+-------------------+------------------+----------------------------+---------------------------+---------------------------------------+
| **value of data** | **size of data** | **value of dataToCompare** | **size of dataToCompare** | **CNM_ReturnTypes.ComparationResult** |
+===================+==================+============================+===========================+=======================================+
| null              | 0                | null                       | 0                         | EQUAL                                 |
+-------------------+------------------+----------------------------+---------------------------+---------------------------------------+
| null              | 0                | 16#01                      | 1                         | SMALLER                               |
+-------------------+------------------+----------------------------+---------------------------+---------------------------------------+
| 16#01             | 1                | null                       | 0                         | GREATER                               |
+-------------------+------------------+----------------------------+---------------------------+---------------------------------------+
| 16#00FF           | 2                | 16#FF                      | 1                         | EQUAL                                 |
+-------------------+------------------+----------------------------+---------------------------+---------------------------------------+
| 16#0100           | 2                | 16#FF                      | 1                         | GREATER                               |
+-------------------+------------------+----------------------------+---------------------------+---------------------------------------+
| 16#FF             | 1                | 16#0100                    | 2                         | SMALLER                               |
+-------------------+------------------+----------------------------+---------------------------+---------------------------------------+
| 16#FF             | 1                | 16#00FF                    | 2                         | EQUAL                                 |
+-------------------+------------------+----------------------------+---------------------------+---------------------------------------+
| 16#0FF0           | 2                | 16#F00F                    | 2                         | SMALLER                               |
+-------------------+------------------+----------------------------+---------------------------+---------------------------------------+

**Attention:** 
	Binary comparison means it compares values byte by byte, regardless of type information (signs, ``REAL`` etc...)
	and it compares padding bytes, too.

**Attention:** 
	``STRING`` and ``WSTRING`` is null terminated
	that means TwinCAT sets null byte/word at the end of the string and touches nothing else
	For example ``foo :STRING(3) := 'foo';`` looks binary 16#66 16#6F 16#6F 16#00.
	if you set foo to an empty string ``foo := ''`` it looks like 16#00 16#6F 16#6F 16#00.

**Attention:** 
	It works not for bits because the minimum size must be at least one byte. If the ``__SYSTEM.TYPE_CLASS``
	of ``data`` ``AND`` ``dataToCompare is ``__SYSTEM.TYPE_CLASS.TYPE_BOOL`` ``OR`` ``__SYSTEM.TYPE_CLASS.TYPE_BIT``
	it uses the ``TO_BOOL`` operator for comarison. That means for ``__SYSTEM.TYPE_CLASS.TYPE_BIT`` it has no idea
	if the single ``BIT`` is set or unset, it compares just the whole ``BYTE``.

.. <legal notes>

legal notes
=================
| SPDX-FileCopyrightText: © 2022 ekvip automation GmbH <info@ekvip.de>
| SPDX-License-Identifier: Apache-2.0
| For details check: Apache-2.0_

.. _Apache-2.0: https://www.apache.org/licenses/LICENSE-2.0

.. </legal notes>


:return: ``SMALLER``: ``data`` is smaller than ``dataToCompare``, 
``EQUAL``: ``data`` is equal to ``dataToCompare``,
``Greater``: ``data`` is greater to ``dataToCompare``

*)

{attribute 'analysis' := '-130'}
METHOD PROTECTED binaryCompare :CNM_ReturnTypes.ComparationResult
VAR_INPUT
	(* current binary data *)
	data			:ANY;
	(* binary data with smaller values *)
	dataToCompare	:ANY;
END_VAR
RETURN(THIS^.isDataNullOrSizeZero(data := data,dataToCompare := dataToCompare,result => binaryCompare));
IF (data.diSize < dataToCompare.diSize) THEN
	IF (THIS^.isDataZero(
		data := dataToCompare.pValue,
		size := dataToCompare.diSize,
		end := dataToCompare.diSize - data.diSize
	)) THEN
		binaryCompare := THIS^.compareData(
			data := data.pValue,
			dataToCompare := dataToCompare.pValue,
			size := data.diSize
		);
	ELSE
		binaryCompare := CNM_ReturnTypes.ComparationResult.SMALLER;
	END_IF
ELSIF (data.diSize > dataToCompare.diSize) THEN
	IF (THIS^.isDataZero(
		data := data.pValue,
		size := data.diSize,
		end := data.diSize - dataToCompare.diSize
	)) THEN
		binaryCompare := THIS^.compareData(
			data := data.pValue,
			dataToCompare := dataToCompare.pValue,
			size := dataToCompare.diSize
		);
	ELSE
		binaryCompare := CNM_ReturnTypes.ComparationResult.GREATER;
	END_IF
ELSIF (THIS^.isDataBoolOrBit(data := data, dataToCompare := dataToCompare)) THEN
	IF (TO_BOOL(data.pValue^) AND (NOT TO_BOOL(dataToCompare.pValue^))) THEN
		binaryCompare := CNM_ReturnTypes.ComparationResult.GREATER;
	ELSIF  ((NOT TO_BOOL(data.pValue^)) AND TO_BOOL(dataToCompare.pValue^)) THEN
		binaryCompare := CNM_ReturnTypes.ComparationResult.SMALLER;
	END_IF
ELSIF (data.diSize = dataToCompare.diSize) THEN
	binaryCompare := THIS^.compareData(
		data := data.pValue,
		dataToCompare := dataToCompare.pValue,
		size := data.diSize
	);
END_IF
END_METHOD

(*

## Short summary
This abstract property returns the class name of the concrete object, 
It's for debugging purpose

.. <legal notes>

legal notes
=================
| SPDX-FileCopyrightText: © 2022 ekvip automation GmbH <info@ekvip.de>
| SPDX-License-Identifier: Apache-2.0
| For details check: Apache-2.0_

.. _Apache-2.0: https://www.apache.org/licenses/LICENSE-2.0

.. </legal notes>

*)

PROPERTY className :CNM_AbstractObject.ClassName
GET
className := 'CNM_Assertor.BinaryAssertions';
END_GET
END_PROPERTY

(*

## Short summary
This method compares the data of two byte pointers. 
The table below shows with some examples how it works.

+-------------------+----------------------------+----------+---------------------------------------+
| **value of data** | **value of dataToCompare** | **size** | **CNM_ReturnTypes.ComparationResult** |
+===================+============================+==========+=======================================+
| 16#00FF           | 16#FF                      | 1        | EQUAL                                 |
+-------------------+----------------------------+----------+---------------------------------------+
| 16#0100           | 16#FF                      | 1        | SMALLER                               |
+-------------------+----------------------------+----------+---------------------------------------+
| 16#FF             | 16#0100                    | 1        | GREATER                               |
+-------------------+----------------------------+----------+---------------------------------------+
| 16#FF             | 16#00FF                    | 1        | EQUAL                                 |
+-------------------+----------------------------+----------+---------------------------------------+
| 16#0FF0           | 16#F00F                    | 1        | GREATER                               |
+-------------------+----------------------------+----------+---------------------------------------+
| 16#0FF0           | 16#F00F                    | 2        | SMALLER                               |
+-------------------+----------------------------+----------+---------------------------------------+

**Attention:** 
	Binary comparison means it compares values byte by byte, regardless of type information (signs, ``REAL`` etc...)
	and it compares padding bytes, too.

**Attention:** 
	``STRING`` and ``WSTRING`` is null terminated
	that means TwinCAT sets null byte/word at the end of the string and touches nothing else
	For example ``foo :STRING(3) := 'foo';`` looks binary 16#66 16#6F 16#6F 16#00.
	if you set foo to an empty string ``foo := ''`` it looks like 16#00 16#6F 16#6F 16#00.

.. <legal notes>

legal notes
=================
| SPDX-FileCopyrightText: © 2022 ekvip automation GmbH <info@ekvip.de>
| SPDX-License-Identifier: Apache-2.0
| For details check: Apache-2.0_

.. _Apache-2.0: https://www.apache.org/licenses/LICENSE-2.0

.. </legal notes>


:return: ``SMALLER``: ``data`` is smaller than ``dataToCompare``, 
``EQUAL``: ``data`` is equal to ``dataToCompare``,
``Greater``: ``data`` is greater to ``dataToCompare``

*)
{attribute 'analysis' := '-41, -130'}
METHOD PROTECTED compareBytewise :CNM_ReturnTypes.ComparationResult
VAR_INPUT
	(* current binary data *)
	data			:POINTER TO BYTE;
	(* current binary data to compare *)
	dataToCompare	:POINTER TO BYTE;
	(* size to compare in bytes, it must be smaller or equal to the smaller size of both data *)
	size			:DINT;
	(* last index to compare *)
	end				:LINT;
END_VAR
VAR
	(* index of the current address *)
	pointerIndex	:LINT;
END_VAR
compareBytewise := CNM_ReturnTypes.ComparationResult.EQUAL;
// memcmp is not used, as it compares from low to highbyte which contradicts the semantics of Numberdatatypes
FOR pointerIndex := (size-1) TO end BY THIS^.DIRECTION_LE DO
	IF (data[pointerIndex] < dataToCompare[pointerIndex]) THEN
		compareBytewise := CNM_ReturnTypes.ComparationResult.SMALLER;
		RETURN;
	ELSIF (data[pointerIndex] > dataToCompare[pointerIndex]) THEN
		compareBytewise := CNM_ReturnTypes.ComparationResult.GREATER;
		RETURN;
	END_IF
END_FOR;
END_METHOD

(*

## Short summary
This method comapres the data of two byte pointers.
It tries to compare registerwise if it makes sens (pointers are aligned and size big enough)
The table below shows with some examples how it works.

+-------------------+------------------+----------------------------+---------------------------+---------------------------------------+
| **value of data** | **size of data** | **value of dataToCompare** | **size of dataToCompare** | **CNM_ReturnTypes.ComparationResult** |
+===================+==================+============================+===========================+=======================================+
| 16#00FF           | 2                | 16#FF                      | 1                         | EQUAL                                 |
+-------------------+------------------+----------------------------+---------------------------+---------------------------------------+
| 16#0100           | 2                | 16#FF                      | 1                         | GREATER                               |
+-------------------+------------------+----------------------------+---------------------------+---------------------------------------+
| 16#FF             | 1                | 16#0100                    | 2                         | SMALLER                               |
+-------------------+------------------+----------------------------+---------------------------+---------------------------------------+
| 16#FF             | 1                | 16#00FF                    | 2                         | EQUAL                                 |
+-------------------+------------------+----------------------------+---------------------------+---------------------------------------+
| 16#0FF0           | 2                | 16#F00F                    | 2                         | SMALLER                               |
+-------------------+------------------+----------------------------+---------------------------+---------------------------------------+

**Attention:** 
	Binary comparison means it compares values byte by byte, regardless of type information (signs, ``REAL`` etc...)
	and it compares padding bytes, too.

**Attention:** 
	``STRING`` and ``WSTRING`` is null terminated
	that means TwinCAT sets null byte/word at the end of the string and touches nothing else
	For example ``foo :STRING(3) := 'foo';`` looks binary 16#66 16#6F 16#6F 16#00.
	if you set foo to an empty string ``foo := ''`` it looks like 16#00 16#6F 16#6F 16#00.

.. <legal notes>

legal notes
=================
| SPDX-FileCopyrightText: © 2022 ekvip automation GmbH <info@ekvip.de>
| SPDX-License-Identifier: Apache-2.0
| For details check: Apache-2.0_

.. _Apache-2.0: https://www.apache.org/licenses/LICENSE-2.0

.. </legal notes>


:return: ``SMALLER``: ``data`` is smaller than ``dataToCompare``, 
``EQUAL``: ``data`` is equal to ``dataToCompare``,
``Greater``: ``data`` is greater to ``dataToCompare``

*)

{attribute 'analysis' := '-130'}
METHOD PROTECTED compareData :CNM_ReturnTypes.ComparationResult
VAR_INPUT
	(* current binary data *)
	data			:POINTER TO BYTE;
	(* current binary data to compare *)
	dataToCompare	:POINTER TO BYTE;
	(* size to compare in bytes, it must be smaller or equal to the smaller size of both data *)
	size			:DINT;
END_VAR
VAR
	(* just a flag to store if both pointer addresses are aligned *)
	arePointersAligned			:BOOL;
	(* number of remaining bytes if it iterates regiterwise through the data*)
	remainingBytes				:DINT;
END_VAR
arePointersAligned := (THIS^.isPointerAligend(data) AND THIS^.isPointerAligend(dataToCompare));

IF (arePointersAligned AND (size >= THIS^.REGISTER_SIZE)) THEN
	remainingBytes := THIS^.getRemainingBytes(size);
	IF (remainingBytes > THIS^.ZERO_SIZE) THEN
		compareData := THIS^.compareBytewise(
			data := data,
			dataToCompare := dataToCompare,
			size := size,
			end := (size - remainingBytes)
		);
		RETURN (compareData <> CNM_ReturnTypes.ComparationResult.EQUAL);
	END_IF
	compareData := THIS^.compareRegisterwise(
		data := data,
		dataToCompare := dataToCompare,
		size := (size - remainingBytes)
	);	
ELSE	
	compareData := THIS^.compareBytewise(
		data := data,
		dataToCompare := dataToCompare,
		size := size,
		end := THIS^.FIRST_DATA
	);
END_IF
END_METHOD

(*

## Short summary
This method comapres the data of two byte pointers, but it iterates registerwise through the data.
The table below shows with some examples how it works.

+------------------------+----------------------------+----------+---------------------------------------+
|    **value of data**   | **value of dataToCompare** | **size** | **CNM_ReturnTypes.ComparationResult** |
+========================+============================+==========+=======================================+
| 16#00FF_FFFF_0000_FFFF | 16#00FF_FFFF_0000_FFFF     | 8        | EQUAL                                 |
+------------------------+----------------------------+----------+---------------------------------------+
| 16#00FF_FFFF_0000_FFFF | 16#80FF_FFFF_0000_FFFF     | 8        | SMALLER                               |
+------------------------+----------------------------+----------+---------------------------------------+
| 16#80FF_FFFF_0000_FFFF | 16#00FF_FFFF_0000_FFFF     | 8        | GREATER                               |
+------------------------+----------------------------+----------+---------------------------------------+
| 16#FFFF_FFFF_0000_FFFF | 16#FFFF_FFFF_0000_FFFF     | 8        | EQUAL                                 |
+------------------------+----------------------------+----------+---------------------------------------+
| 16#80FF_FFFF_0000_FFFF | 16#70FF_FFFF_FFFF_FFFF     | 8        | GREATER                               |
+------------------------+----------------------------+----------+---------------------------------------+
| 16#70FF_FFFF_FFFF_FFFF | 16#80FF_FFFF_0000_FFFF     | 8        | SMALLER                               |
+------------------------+----------------------------+----------+---------------------------------------+

**Attention:** 
	Binary comparison means it compares values register by register, regardless of type information (signs, ``REAL`` etc...)
	and it compares padding bytes, too.

**Attention:** 
	``STRING`` and ``WSTRING`` is null terminated
	that means TwinCAT sets null byte/word at the end of the string and touches nothing else
	For example ``foo :STRING(3) := 'foo';`` looks binary 16#66 16#6F 16#6F 16#00.
	if you set foo to an empty string ``foo := ''`` it looks like 16#00 16#6F 16#6F 16#00.

.. <legal notes>

legal notes
=================
| SPDX-FileCopyrightText: © 2022 ekvip automation GmbH <info@ekvip.de>
| SPDX-License-Identifier: Apache-2.0
| For details check: Apache-2.0_

.. _Apache-2.0: https://www.apache.org/licenses/LICENSE-2.0

.. </legal notes>


:return: ``SMALLER``: ``data`` is smaller than ``dataToCompare``, 
``EQUAL``: ``data`` is equal to ``dataToCompare``,
``Greater``: ``data`` is greater to ``dataToCompare``

*)

{attribute 'analysis' := '-41, -130'}
METHOD PROTECTED compareRegisterwise :CNM_ReturnTypes.ComparationResult
VAR_INPUT
	(* current binary data *)
	data			:POINTER TO __XWORD;
	(* current binary data to compare *)
	dataToCompare	:POINTER TO __XWORD;
	(* size to compare in bytes, size must be a muliple of register size *)
	size			:DINT;
END_VAR
VAR
	(* index of the current address *)
	pointerIndex	:LINT;
END_VAR
compareRegisterwise := CNM_ReturnTypes.ComparationResult.EQUAL;

FOR pointerIndex := (((size)/THIS^.REGISTER_SIZE)-1) TO THIS^.FIRST_DATA BY THIS^.DIRECTION_LE DO
	IF (data[pointerIndex] < dataToCompare[pointerIndex]) THEN
		compareRegisterwise := CNM_ReturnTypes.ComparationResult.SMALLER;
		RETURN;
	ELSIF (data[pointerIndex] > dataToCompare[pointerIndex]) THEN
		compareRegisterwise := CNM_ReturnTypes.ComparationResult.GREATER;
		RETURN;
	END_IF
END_FOR;
END_METHOD

(*

## Short summary
This method calculates the number of bytes that are remaining
if size is divided by register size.

.. <legal notes>

legal notes
=================
| SPDX-FileCopyrightText: © 2022 ekvip automation GmbH <info@ekvip.de>
| SPDX-License-Identifier: Apache-2.0
| For details check: Apache-2.0_

.. _Apache-2.0: https://www.apache.org/licenses/LICENSE-2.0

.. </legal notes>


:return: number of bytes that are remaining if it iterates registerwise through the data

*)

METHOD PROTECTED getRemainingBytes :DINT
VAR_INPUT
	(* size in bytes *)
	size			:DINT;
END_VAR
getRemainingBytes := (size MOD THIS^.REGISTER_SIZE);
END_METHOD

(*

## Short summary
This method checks if the current Data and DataToCompare are both either bools or bits.

.. <legal notes>

legal notes
=================
| SPDX-FileCopyrightText: © 2022 ekvip automation GmbH <info@ekvip.de>
| SPDX-License-Identifier: Apache-2.0
| For details check: Apache-2.0_

.. _Apache-2.0: https://www.apache.org/licenses/LICENSE-2.0

.. </legal notes>


:return: ``TRUE`` data and dataToCompare are both bool / bits, otherwise false

*)

METHOD PROTECTED isDataBoolOrBit : BOOL
VAR_INPUT
	(* current binary data *)
	data			:ANY;
	(* binary data with smaller values *)
	dataToCompare	:ANY;
END_VAR
VAR CONSTANT
	(* for boolens to figure out if the size exactly one byte *) 
	SIZE_OF_ONE_BYTE	:DINT := 1;
END_VAR
isDataBoolOrBit := ((
	data.diSize = SIZE_OF_ONE_BYTE
	) AND (
		dataToCompare.diSize = SIZE_OF_ONE_BYTE
	) AND ( 
		(data.TypeClass = TYPE_CLASS.TYPE_BOOL)
		OR 	(data.TypeClass = TYPE_CLASS.TYPE_BIT)
	) AND (
			(dataToCompare.TypeClass = TYPE_CLASS.TYPE_BOOL)
			OR (dataToCompare.TypeClass = TYPE_CLASS.TYPE_BIT)
	)
);
END_METHOD

(*

## Short summary
This method checks if the two given pointers have a valid address and the size of data is defined.

+-------------------+------------------+----------------------------+---------------------------+---------------------------------------+--------------------------+
| **value of data** | **size of data** | **value of dataToCompare** | **size of dataToCompare** | **CNM_ReturnTypes.ComparationResult** | **ReturnValue**		   |
+===================+==================+============================+===========================+=======================================+==========================+
| null              | *                | null                       | *                         | EQUAL                                 | TRUE					   |
+-------------------+------------------+----------------------------+---------------------------+---------------------------------------+--------------------------+
| *              	| 0                | *	                        | 0                         | EQUAL                                 | TRUE					   |
+-------------------+------------------+----------------------------+---------------------------+---------------------------------------+--------------------------+
| null              | *                | *                          | *                         | SMALLER                               | TRUE					   |
+-------------------+------------------+----------------------------+---------------------------+---------------------------------------+--------------------------+
| *                 | 0                | *                          | *                         | SMALLER                               | TRUE					   |
+-------------------+------------------+----------------------------+---------------------------+---------------------------------------+--------------------------+
| *                 | *                | null                       | *                         | GREATER                               | TRUE					   |
+-------------------+------------------+----------------------------+---------------------------+---------------------------------------+--------------------------+
| *                 | *                | *                          | 0                         | GREATER                               | TRUE					   |
+-------------------+------------------+----------------------------+---------------------------+---------------------------------------+--------------------------+
Otherwise: EQUAL, FALSE
( referes to something not null / <> 0)


legal notes
=================
| SPDX-FileCopyrightText: © 2025 ekvip automation GmbH <info@ekvip.de>
| SPDX-License-Identifier: Apache-2.0
| For details check: Apache-2.0_

.. _Apache-2.0: https://www.apache.org/licenses/LICENSE-2.0

.. </legal notes>


:return: consider table

*)

METHOD PROTECTED isDataNullOrSizeZero : BOOL
VAR_INPUT
	(* current binary data *)
	data			:ANY;
	(* binary data with smaller values *)
	dataToCompare	:ANY;
END_VAR
VAR_OUTPUT
	(*see table*)
	result: CNM_ReturnTypes.ComparationResult;
END_VAR
result := CNM_ReturnTypes.ComparationResult.EQUAL;
isDataNullOrSizeZero := TRUE;
RETURN ((data.pValue = THIS^.NULL_POINTER) AND (dataToCompare.pValue = THIS^.NULL_POINTER));
RETURN ((data.diSize = THIS^.ZERO_SIZE) AND (dataToCompare.diSize = THIS^.ZERO_SIZE));
IF (
	((data.pValue = THIS^.NULL_POINTER) AND (dataToCompare.pValue <> THIS^.NULL_POINTER))
	OR ((data.diSize = THIS^.ZERO_SIZE) AND (dataToCompare.diSize <> THIS^.ZERO_SIZE))
)THEN
	result := CNM_ReturnTypes.ComparationResult.SMALLER;
ELSIF (
	((data.pValue <> THIS^.NULL_POINTER) AND (dataToCompare.pValue = THIS^.NULL_POINTER))
	OR ((data.diSize <> THIS^.ZERO_SIZE) AND (dataToCompare.diSize = THIS^.ZERO_SIZE))
)THEN
	result := CNM_ReturnTypes.ComparationResult.GREATER;
ELSE
	isDataNullOrSizeZero := FALSE;
END_IF;
END_METHOD

(*

## Short summary
This method checks if the data of a pointer is zero through all bytes (``size-1``)

+------------------------+----------+---------+------------------+
|    **value of data**   | **size** | **end** | **return value** |
+========================+==========+=========+==================+
| 16#00FF_FFFF_0000_0000 | 8        | 7       | TRUE             |
+------------------------+----------+---------+------------------+
| 16#00FF_FFFF_0000_0000 | 8        | 6       | FALSE            |
+------------------------+----------+---------+------------------+
| 16#80FF_FFFF_0000_0000 | 8        | 7       | FALSE            |
+------------------------+----------+---------+------------------+
| 16#0000_0000_0000_FFFF | 8        | 2       | TRUE             |
+------------------------+----------+---------+------------------+
| 16#0000_0000_0000_FFFF | 8        | 1       | FALSE            |
+------------------------+----------+---------+------------------+
| 16#70FF_FFFF_FFFF_FFFF | 8        | 8       | TRUE             |
+------------------------+----------+---------+------------------+

.. <legal notes>

legal notes
=================
| SPDX-FileCopyrightText: © 2022 ekvip automation GmbH <info@ekvip.de>
| SPDX-License-Identifier: Apache-2.0
| For details check: Apache-2.0_

.. _Apache-2.0: https://www.apache.org/licenses/LICENSE-2.0

.. </legal notes>


:return: ``TRUE`` all bytes are zero, ``FALSE`` at least one byte isn't zero

*)

{attribute 'analysis' := '-130'}
METHOD PROTECTED isDataZero :BOOL
VAR_INPUT
	(* current binary data *)
	data			:POINTER TO BYTE;
	(* size to compare in bytes *)
	size			:DINT;
	(* last index to compare *)
	end				:LINT;	
END_VAR
VAR
	isPointerAligned			:BOOL;
	remainingBytes				:DINT;
END_VAR
isPointerAligned := THIS^.isPointerAligend(data);

IF (isPointerAligned AND_THEN ((size-end) >= THIS^.REGISTER_SIZE)) THEN
	remainingBytes := THIS^.getRemainingBytes(size);
	IF (remainingBytes > THIS^.ZERO_SIZE) THEN
		isDataZero := THIS^.isDataZeroBytewise(
			data := data,
			size := size,
			end := (size - remainingBytes)
		);
		RETURN (NOT isDataZero);
	END_IF
	isDataZero := THIS^.isDataZeroRegisterwise(
		data := data,
		size := (size - remainingBytes),
		end := end
	);	
ELSE	
	isDataZero := THIS^.isDataZeroBytewise(
		data := data,
		size := size,
		end := end
	);
END_IF;
END_METHOD

(*

## Short summary
This method checks if the data of a byte pointer is zero through all bytes form (``size-1``) to ``end``.
The table below shows how it works.

+------------------------+----------+---------+------------------+
|    **value of data**   | **size** | **end** | **return value** |
+========================+==========+=========+==================+
| 16#00FF_FFFF_0000_0000 | 8        | 7       | TRUE             |
+------------------------+----------+---------+------------------+
| 16#00FF_FFFF_0000_0000 | 8        | 6       | FALSE            |
+------------------------+----------+---------+------------------+
| 16#80FF_FFFF_0000_0000 | 8        | 7       | FALSE            |
+------------------------+----------+---------+------------------+
| 16#0000_0000_0000_FFFF | 8        | 2       | TRUE             |
+------------------------+----------+---------+------------------+
| 16#0000_0000_0000_FFFF | 8        | 1       | FALSE            |
+------------------------+----------+---------+------------------+
| 16#70FF_FFFF_FFFF_FFFF | 8        | 8       | TRUE             |
+------------------------+----------+---------+------------------+

.. <legal notes>

legal notes
=================
| SPDX-FileCopyrightText: © 2022 ekvip automation GmbH <info@ekvip.de>
| SPDX-License-Identifier: Apache-2.0
| For details check: Apache-2.0_

.. _Apache-2.0: https://www.apache.org/licenses/LICENSE-2.0

.. </legal notes>


:return: ``TRUE`` all bytes are zero, ``FALSE`` at least one byte isn't zero

*)

{attribute 'analysis' := '-130, -41'}
METHOD PROTECTED isDataZeroBytewise :BOOL
VAR_INPUT
	(* current binary data *)
	data			:POINTER TO BYTE;
	(* size to compare in bytes *)
	size			:DINT;
	(* last index to compare *)
	end				:LINT;
END_VAR
VAR
	(* index of the current address *)
	pointerIndex	:LINT;
END_VAR
VAR CONSTANT
	NULL			:BYTE := 16#00;
END_VAR
isDataZeroBytewise := TRUE;

FOR pointerIndex := (size-1) TO end BY THIS^.DIRECTION_LE DO
	IF (data[pointerIndex] <> NULL) THEN
		isDataZeroBytewise := FALSE;
		RETURN;
	END_IF
END_FOR;
END_METHOD

(*

## Short summary
This method checks if the data of a ``__XWORD pointer`` is zero
through all bytes form (``size-1``) to ``end``.

.. <legal notes>

legal notes
=================
| SPDX-FileCopyrightText: © 2022 ekvip automation GmbH <info@ekvip.de>
| SPDX-License-Identifier: Apache-2.0
| For details check: Apache-2.0_

.. _Apache-2.0: https://www.apache.org/licenses/LICENSE-2.0

.. </legal notes>


:return: ``TRUE`` all bytes are zero, ``FALSE`` at least one byte isn't zero

*)

{attribute 'analysis' := '-41, -130'}
METHOD PROTECTED isDataZeroRegisterwise :BOOL
VAR_INPUT
	(* current binary data *)
	data			:POINTER TO __XWORD;
	(* size to compare in bytes *)
	size			:DINT;
	(* last index to compare *)
	end				:LINT;
END_VAR
VAR
	(* index of the current address *)
	pointerIndex	:LINT;
END_VAR
VAR CONSTANT
	NULL			:__XWORD := 0;
END_VAR
isDataZeroRegisterwise := TRUE;

FOR pointerIndex := (size-1) TO end BY THIS^.DIRECTION_LE DO
	IF (data[pointerIndex] <> NULL) THEN
		isDataZeroRegisterwise := FALSE;
		RETURN;
	END_IF
END_FOR;
END_METHOD

(*

## Short summary
This assertion method checks if all bytes of memory of
``data`` and ``dataToCompare`` are equal

**Attention:** 
	Binary comparison means it compares values byte by byte, regardless of type information (signs, ``REAL`` etc...)
	and it compares padding bytes, too.

**Attention:** 
	``STRING`` and ``WSTRING`` is null terminated
	that means TwinCAT sets null byte/word at the end of the string and touches nothing else
	For example ``foo :STRING(3) := 'foo';`` looks binary 16#66 16#6F 16#6F 16#00.
	if you set foo to an empty string ``foo := ''`` it looks like 16#00 16#6F 16#6F 16#00.

**Attention:** 
	It works not for bits because the minimum size must be at least one byte. If the ``__SYSTEM.TYPE_CLASS``
	of ``data`` ``AND`` ``dataToCompare is ``__SYSTEM.TYPE_CLASS.TYPE_BOOL`` ``OR`` ``__SYSTEM.TYPE_CLASS.TYPE_BIT``
	it uses the ``TO_BOOL`` operator for comarison. That means for ``__SYSTEM.TYPE_CLASS.TYPE_BIT`` it has no idea
	if the single ``BIT`` is set or unset, it compares just the whole ``BYTE``.

.. <legal notes>

legal notes
=================
| SPDX-FileCopyrightText: © 2022 ekvip automation GmbH <info@ekvip.de>
| SPDX-License-Identifier: Apache-2.0
| For details check: Apache-2.0_

.. _Apache-2.0: https://www.apache.org/licenses/LICENSE-2.0

.. </legal notes>



*)

METHOD isEqualTo
VAR_INPUT
	(* current binary data *)
	data			:ANY;
	(* binary data with the expected values *)
	dataToCompare	:ANY;
	(* message if the assertion is false *)
	message			:AssertMessage;
END_VAR
IF (THIS^.binaryCompare(data, dataToCompare) <> CNM_ReturnTypes.ComparationResult.EQUAL) THEN
	THIS^.assertionWasWrong(message, THIS^.getDebugInfo('isEqualTo'));
END_IF
END_METHOD

(*

## Short summary
This assertion method checks the bytes of memory of
``data`` and ``dataToCompare`` if the content of the first unequal
``data`` byte is greater than the byte of ``dataToCompare``
the assertion is true. Direction of comaprison is little endian.

**Attention:** 
	Binary comparison means it compares values byte by byte, regardless of type information (signs, ``REAL`` etc...)
	and it compares padding bytes, too.

**Attention:** 
	``STRING`` and ``WSTRING`` is null terminated
	that means TwinCAT sets null byte/word at the end of the string and touches nothing else
	For example ``foo :STRING(3) := 'foo';`` looks binary 16#66 16#6F 16#6F 16#00.
	if you set foo to an empty string ``foo := ''`` it looks like 16#00 16#6F 16#6F 16#00.

**Attention:** 
	It works not for bits because the minimum size must be at least one byte. If the ``__SYSTEM.TYPE_CLASS``
	of ``data`` ``AND`` ``dataToCompare is ``__SYSTEM.TYPE_CLASS.TYPE_BOOL`` ``OR`` ``__SYSTEM.TYPE_CLASS.TYPE_BIT``
	it uses the ``TO_BOOL`` operator for comarison. That means for ``__SYSTEM.TYPE_CLASS.TYPE_BIT`` it has no idea
	if the single ``BIT`` is set or unset, it compares just the whole ``BYTE``.

.. <legal notes>

legal notes
=================
| SPDX-FileCopyrightText: © 2022 ekvip automation GmbH <info@ekvip.de>
| SPDX-License-Identifier: Apache-2.0
| For details check: Apache-2.0_

.. _Apache-2.0: https://www.apache.org/licenses/LICENSE-2.0

.. </legal notes>



*)

METHOD isGreaterThan
VAR_INPUT
	(* current binary data *)
	data			:ANY;
	(* binary data with smaller values *)
	dataToCompare	:ANY;
	(* message if the assertion is false *)
	message			:AssertMessage;
END_VAR
IF (THIS^.binaryCompare(data, dataToCompare) <> CNM_ReturnTypes.ComparationResult.GREATER) THEN
	THIS^.assertionWasWrong(message, THIS^.getDebugInfo('isGreaterThan'));
END_IF
END_METHOD

(*

## Short summary
This assertion method checks the bytes of memory of
``data`` and ``dataToCompare`` if the content of the first unequal
``data`` byte is less than the byte of ``dataToCompare``
the assertion is true. Direction of comaprison is little endian.

.. <legal notes>

**Attention:** 
	Binary comparison means it compares values byte by byte, regardless of type information (signs, ``REAL`` etc...)
	and it compares padding bytes, too.

**Attention:** 
	``STRING`` and ``WSTRING`` is null terminated
	that means TwinCAT sets null byte/word at the end of the string and touches nothing else
	For example ``foo :STRING(3) := 'foo';`` looks binary 16#66 16#6F 16#6F 16#00.
	if you set foo to an empty string ``foo := ''`` it looks like 16#00 16#6F 16#6F 16#00.

**Attention:** 
	It works not for bits because the minimum size must be at least one byte. If the ``__SYSTEM.TYPE_CLASS``
	of ``data`` ``AND`` ``dataToCompare is ``__SYSTEM.TYPE_CLASS.TYPE_BOOL`` ``OR`` ``__SYSTEM.TYPE_CLASS.TYPE_BIT``
	it uses the ``TO_BOOL`` operator for comarison. That means for ``__SYSTEM.TYPE_CLASS.TYPE_BIT`` it has no idea
	if the single ``BIT`` is set or unset, it compares just the whole ``BYTE``.

legal notes
=================
| SPDX-FileCopyrightText: © 2022 ekvip automation GmbH <info@ekvip.de>
| SPDX-License-Identifier: Apache-2.0
| For details check: Apache-2.0_

.. _Apache-2.0: https://www.apache.org/licenses/LICENSE-2.0

.. </legal notes>



*)

METHOD isLessThan
VAR_INPUT
	(* current binary data *)
	data			:ANY;
	(* binary data with greater values *)
	dataToCompare	:ANY;
	(* message if the assertion is false *)
	message			:AssertMessage;
END_VAR
IF (THIS^.binaryCompare(data, dataToCompare) <> CNM_ReturnTypes.ComparationResult.SMALLER) THEN
	THIS^.assertionWasWrong(message, THIS^.getDebugInfo('isLessThan'));
END_IF
END_METHOD

(*

## Short summary
This assertion method checks if minimal one byte of memory of
``data`` and ``dataToCompare`` is not equal

**Attention:** 
	Binary comparison means it compares values byte by byte, regardless of type information (signs, ``REAL`` etc...)
	and it compares padding bytes, too.

**Attention:** 
	``STRING`` and ``WSTRING`` is null terminated
	that means TwinCAT sets null byte/word at the end of the string and touches nothing else
	For example ``foo :STRING(3) := 'foo';`` looks binary 16#66 16#6F 16#6F 16#00.
	if you set foo to an empty string ``foo := ''`` it looks like 16#00 16#6F 16#6F 16#00.

**Attention:** 
	It works not for bits because the minimum size must be at least one byte. If the ``__SYSTEM.TYPE_CLASS``
	of ``data`` ``AND`` ``dataToCompare is ``__SYSTEM.TYPE_CLASS.TYPE_BOOL`` ``OR`` ``__SYSTEM.TYPE_CLASS.TYPE_BIT``
	it uses the ``TO_BOOL`` operator for comarison. That means for ``__SYSTEM.TYPE_CLASS.TYPE_BIT`` it has no idea
	if the single ``BIT`` is set or unset, it compares just the whole ``BYTE``.

.. <legal notes>

legal notes
=================
| SPDX-FileCopyrightText: © 2022 ekvip automation GmbH <info@ekvip.de>
| SPDX-License-Identifier: Apache-2.0
| For details check: Apache-2.0_

.. _Apache-2.0: https://www.apache.org/licenses/LICENSE-2.0

.. </legal notes>



*)

METHOD isNotEqualTo
VAR_INPUT
	(* current binary data *)
	data			:ANY;
	(* binary data with the unexpected values *)
	dataToCompare	:ANY;
	(* message if the assertion is false *)
	message			:AssertMessage;
END_VAR
IF (THIS^.binaryCompare(data, dataToCompare) = CNM_ReturnTypes.ComparationResult.EQUAL) THEN
	THIS^.assertionWasWrong(message, THIS^.getDebugInfo('isNotEqualTo'));
END_IF
END_METHOD

(*

## Short summary
This method checks if an address is aligned to a register

.. <legal notes>

legal notes
=================
| SPDX-FileCopyrightText: © 2022 ekvip automation GmbH <info@ekvip.de>
| SPDX-License-Identifier: Apache-2.0
| For details check: Apache-2.0_

.. _Apache-2.0: https://www.apache.org/licenses/LICENSE-2.0

.. </legal notes>


:return: ``TRUE`` pointer address **is** aligned to a register,
``FALSE`` pointer address **isn't** aligned to a register

*)

METHOD PROTECTED isPointerAligend :BOOL
VAR_INPUT
	(* address to check *)
	in :PVOID;
END_VAR
VAR CONSTANT
	(* 
	for 32 bit systems address is aligned if 2#111 is unset,
	for 64 bit systems address is aligned if 2#1111 is unset
	*)
	ALIGNMENT_MASK	:__XWORD := (SIZEOF(__XWORD)-1);
	(* just to check if relevant bits unset *)
	WELL_ALIGNED	:__XWORD := 0;
END_VAR
isPointerAligend := ((in AND ALIGNMENT_MASK) = WELL_ALIGNED);
END_METHOD

END_FUNCTION_BLOCK

// ---- Assertor/classes/AbstractAssertion.TcPOU
(*

## Short summary
This abstract class is for all the assertion classes to ease and unify
the callbacks

.. <legal notes>

legal notes
=================
| SPDX-FileCopyrightText: © 2022 ekvip automation GmbH <info@ekvip.de>
| SPDX-License-Identifier: Apache-2.0
| For details check: Apache-2.0_

.. _Apache-2.0: https://www.apache.org/licenses/LICENSE-2.0

.. </legal notes>



*)

{attribute 'reflection'}
FUNCTION_BLOCK INTERNAL ABSTRACT AbstractAssertion EXTENDS CNM_AbstractObject.Object IMPLEMENTS IAssertCallBackSetter
VAR
	(* the class that must be informed if an assertion is false *)
	callBack	:IAssertCallBack;
END_VAR

(*

## Short summary
This method is called if an assertion was ``FALSE``

.. <legal notes>

legal notes
=================
| SPDX-FileCopyrightText: © 2022 ekvip automation GmbH <info@ekvip.de>
| SPDX-License-Identifier: Apache-2.0
| For details check: Apache-2.0_

.. _Apache-2.0: https://www.apache.org/licenses/LICENSE-2.0

.. </legal notes>



*)

METHOD PROTECTED assertionWasWrong
VAR_INPUT
	(* alarm message *)
	message			:AssertMessage;
	(* debugging information *) 
	additionalText	:Tc2_System.T_MaxString;
END_VAR
IF (THIS^.isObjectValid(THIS^.callBack)) THEN
	THIS^.callBack.assertionWasWrong(
		caller			:= THIS^,
		message			:= message,
		additionalText	:= additionalText
	);
END_IF
END_METHOD

(*

## Short summary
This abstract property returns the class name of the concrete object, 
It's for debugging purpose

**Attention:** 
	For derivations: **It is necessary that this property is overridden by the concrete class**

.. <legal notes>

legal notes
=================
| SPDX-FileCopyrightText: © 2022 ekvip automation GmbH <info@ekvip.de>
| SPDX-License-Identifier: Apache-2.0
| For details check: Apache-2.0_

.. _Apache-2.0: https://www.apache.org/licenses/LICENSE-2.0

.. </legal notes>

*)

PROPERTY ABSTRACT className : CNM_AbstractObject.ClassName
GET
END_GET
END_PROPERTY

(*

## Short summary
This method returns a debug info string

.. <legal notes>

legal notes
=================
| SPDX-FileCopyrightText: © 2022 ekvip automation GmbH <info@ekvip.de>
| SPDX-License-Identifier: Apache-2.0
| For details check: Apache-2.0_

.. _Apache-2.0: https://www.apache.org/licenses/LICENSE-2.0

.. </legal notes>


:return: debug info string, it contains the caller method name and the class name. 
Format is ``'ClassName.methodName: Assertion was false'``

*)

METHOD PROTECTED getDebugInfo :Tc2_System.T_MaxString
VAR_INPUT
	(* name of the caller method *) 
	caller	:Tc2_System.T_MaxString;
END_VAR
getDebugInfo := Tc2_Standard.CONCAT(
	THIS^.className,
	Tc2_Standard.CONCAT(
		'.',
		Tc2_Standard.CONCAT(
			caller,
			': Assertion was false'
		)
	)
);
END_METHOD

(*

## Short summary
This methods is the setter for the callback class if an assertion was false

.. <legal notes>

legal notes
=================
| SPDX-FileCopyrightText: © 2022 ekvip automation GmbH <info@ekvip.de>
| SPDX-License-Identifier: Apache-2.0
| For details check: Apache-2.0_

.. _Apache-2.0: https://www.apache.org/licenses/LICENSE-2.0

.. </legal notes>



*)

METHOD setCallBack
VAR_INPUT
	(* the class that must be informed if an assertion is false *)
	callBack	:IAssertCallBack;  
END_VAR
THIS^.callBack := callBack;
END_METHOD

END_FUNCTION_BLOCK

// ---- Assertor/Assertions/BitNumberAssertions/Byte/classes/ByteAssertions.TcPOU
(*

## Short summary
This class provides assert statements for bytes.

.. <legal notes>

legal notes
=================
| SPDX-FileCopyrightText: © 2022 ekvip automation GmbH <info@ekvip.de>
| SPDX-License-Identifier: Apache-2.0
| For details check: Apache-2.0_

.. _Apache-2.0: https://www.apache.org/licenses/LICENSE-2.0

.. </legal notes>



*)

{attribute 'reflection'}
FUNCTION_BLOCK INTERNAL ByteAssertions EXTENDS AbstractAssertion IMPLEMENTS IByteAssertions
VAR
END_VAR
VAR CONSTANT
	(* least significant bit *)
	LSB	:BYTE := 16#01;
	(* most significant bit *)
	MSB :BYTE := 16#80;
END_VAR

(*

## Short summary
This assertion method checks if the result current value bitwise ``AND`` mask is equal to the expected value

.. <legal notes>

legal notes
=================
| SPDX-FileCopyrightText: © 2022 ekvip automation GmbH <info@ekvip.de>
| SPDX-License-Identifier: Apache-2.0
| For details check: Apache-2.0_

.. _Apache-2.0: https://www.apache.org/licenses/LICENSE-2.0

.. </legal notes>



*)

METHOD andMaskIsEqualTo
VAR_INPUT
	(* current value to check *)
	currentValue	:BYTE;
	(* 2nd operand for bitwise operation *)
	mask			:BYTE;
	(* expected result after masking *)
	expectedValue	:BYTE;
	(* message if the assertion is false *)
	message			:AssertMessage;
END_VAR
IF ((currentValue AND mask) <> expectedValue) THEN
	THIS^.assertionWasWrong(message, THIS^.getDebugInfo('andMaskIsEqualTo'));
END_IF
END_METHOD

(*

## Short summary
This assertion method checks if the result current value bitwise ``AND`` mask
is not equal to the unexpected value

.. <legal notes>

legal notes
=================
| SPDX-FileCopyrightText: © 2022 ekvip automation GmbH <info@ekvip.de>
| SPDX-License-Identifier: Apache-2.0
| For details check: Apache-2.0_

.. _Apache-2.0: https://www.apache.org/licenses/LICENSE-2.0

.. </legal notes>



*)

METHOD andMaskIsNotEqualTo
VAR_INPUT
	(* current value to check *)
	currentValue	:BYTE;
	(* 2nd operand for bitwise operation *)
	mask			:BYTE;
	(* unexpected result after masking *)
	unexpectedValue	:BYTE;
	(* message if the assertion is false *)
	message			:AssertMessage;
END_VAR
IF ((currentValue AND mask) = unexpectedValue) THEN
	THIS^.assertionWasWrong(message, THIS^.getDebugInfo('andMaskIsNotEqualTo'));
END_IF
END_METHOD

(*

## Short summary
This assertion method checks if the selected bit of current value
is equal to the expected value

.. <legal notes>

legal notes
=================
| SPDX-FileCopyrightText: © 2022 ekvip automation GmbH <info@ekvip.de>
| SPDX-License-Identifier: Apache-2.0
| For details check: Apache-2.0_

.. _Apache-2.0: https://www.apache.org/licenses/LICENSE-2.0

.. </legal notes>



*)

METHOD bitXIsEqualTo
VAR_INPUT
	(* current value to check *)
	currentValue	:BYTE;
	(* number of bit to check *)
	number			:BitNumberByte;
	(* expected value of bit *)
	expectedValue	:BOOL;
	(* message if the assertion is false *)
	message			:AssertMessage;
END_VAR
IF (
	TO_BOOL(
		TO_BYTE(SHL(THIS^.LSB, number))
		AND currentValue
	) <> expectedValue
) THEN
	THIS^.assertionWasWrong(message, THIS^.getDebugInfo('bitXIsEqualTo'));
END_IF
END_METHOD

(*

## Short summary
This assertion method checks if the selected bit of current value
is not equal to the unexpected value

.. <legal notes>

legal notes
=================
| SPDX-FileCopyrightText: © 2022 ekvip automation GmbH <info@ekvip.de>
| SPDX-License-Identifier: Apache-2.0
| For details check: Apache-2.0_

.. _Apache-2.0: https://www.apache.org/licenses/LICENSE-2.0

.. </legal notes>



*)

METHOD bitXIsNotEqualTo
VAR_INPUT
	(* current value to check *)
	currentValue	:BYTE;
	(* number of bit to check *)
	number			:BitNumberByte;
	(* unexpected value of bit *)
	unexpectedValue	:BOOL;
	(* message if the assertion is false *)
	message			:AssertMessage;
END_VAR
IF (
	TO_BOOL(
		TO_BYTE(SHL(THIS^.LSB, number))
		AND currentValue
	) = unexpectedValue
) THEN
	THIS^.assertionWasWrong(message, THIS^.getDebugInfo('bitXIsNotEqualTo'));
END_IF
END_METHOD

(*

## Short summary
This assertion method checks if the selected bit of current value
is set

.. <legal notes>

legal notes
=================
| SPDX-FileCopyrightText: © 2022 ekvip automation GmbH <info@ekvip.de>
| SPDX-License-Identifier: Apache-2.0
| For details check: Apache-2.0_

.. _Apache-2.0: https://www.apache.org/licenses/LICENSE-2.0

.. </legal notes>



*)

METHOD bitXIsSet
VAR_INPUT
	(* current value to check *)
	currentValue	:BYTE;
	(* number of bit to check *)
	number			:BitNumberByte;
	(* message if the assertion is false *)
	message			:AssertMessage;
END_VAR
IF (
	NOT TO_BOOL(
		TO_BYTE(SHL(THIS^.LSB, number))
		AND currentValue
	)
) THEN
	THIS^.assertionWasWrong(message, THIS^.getDebugInfo('bitXIsSet'));
END_IF
END_METHOD

(*

## Short summary
This assertion method checks if the selected bit of current value
is unset

.. <legal notes>

legal notes
=================
| SPDX-FileCopyrightText: © 2022 ekvip automation GmbH <info@ekvip.de>
| SPDX-License-Identifier: Apache-2.0
| For details check: Apache-2.0_

.. _Apache-2.0: https://www.apache.org/licenses/LICENSE-2.0

.. </legal notes>



*)

METHOD bitXIsUnset
VAR_INPUT
	(* current value to check *)
	currentValue	:BYTE;
	(* number of bit to check *)
	number			:BitNumberByte;
	(* message if the assertion is false *)
	message			:AssertMessage;
END_VAR
IF (
	TO_BOOL(
		TO_BYTE(SHL(THIS^.LSB, number))
		AND currentValue
	)
) THEN
	THIS^.assertionWasWrong(message, THIS^.getDebugInfo('bitXIsUnset'));
END_IF
END_METHOD

(*

## Short summary
This abstract property returns the class name of the concrete object, 
It's for debugging purpose

.. <legal notes>

legal notes
=================
| SPDX-FileCopyrightText: © 2022 ekvip automation GmbH <info@ekvip.de>
| SPDX-License-Identifier: Apache-2.0
| For details check: Apache-2.0_

.. _Apache-2.0: https://www.apache.org/licenses/LICENSE-2.0

.. </legal notes>

*)

PROPERTY className :CNM_AbstractObject.ClassName
GET
className := 'CNM_Assertor.ByteAssertions';
END_GET
END_PROPERTY

(*

## Short summary
This assertion method checks if the least significant bit of current value
is equal to the expected value

.. <legal notes>

legal notes
=================
| SPDX-FileCopyrightText: © 2022 ekvip automation GmbH <info@ekvip.de>
| SPDX-License-Identifier: Apache-2.0
| For details check: Apache-2.0_

.. _Apache-2.0: https://www.apache.org/licenses/LICENSE-2.0

.. </legal notes>



*)

METHOD lsbIsEqualTo
VAR_INPUT
	(* current value to check *)
	currentValue	:BYTE;
	(* expected value of lsb *)
	expectedValue	:BOOL;
	(* message if the assertion is false *)
	message			:AssertMessage;
END_VAR
IF (TO_BOOL(currentValue AND THIS^.LSB) <> expectedValue) THEN
	THIS^.assertionWasWrong(message, THIS^.getDebugInfo('lsbIsEqualTo'));
END_IF
END_METHOD

(*

## Short summary
This assertion method checks if the least significant bit of current value
is not equal to the unexpected value

.. <legal notes>

legal notes
=================
| SPDX-FileCopyrightText: © 2022 ekvip automation GmbH <info@ekvip.de>
| SPDX-License-Identifier: Apache-2.0
| For details check: Apache-2.0_

.. _Apache-2.0: https://www.apache.org/licenses/LICENSE-2.0

.. </legal notes>



*)

METHOD lsbIsNotEqualTo
VAR_INPUT
	(* current value to check *)
	currentValue	:BYTE;
	(* unexpected value of lsb *)
	unexpectedValue	:BOOL;
	(* message if the assertion is false *)
	message			:AssertMessage;
END_VAR
IF (TO_BOOL(currentValue AND THIS^.LSB) = unexpectedValue) THEN
	THIS^.assertionWasWrong(message, THIS^.getDebugInfo('lsbIsNotEqualTo'));
END_IF
END_METHOD

(*

## Short summary
This assertion method checks if the least significant bit of current value
is set

.. <legal notes>

legal notes
=================
| SPDX-FileCopyrightText: © 2022 ekvip automation GmbH <info@ekvip.de>
| SPDX-License-Identifier: Apache-2.0
| For details check: Apache-2.0_

.. _Apache-2.0: https://www.apache.org/licenses/LICENSE-2.0

.. </legal notes>



*)

METHOD lsbIsSet
VAR_INPUT
	(* current value to check *)
	currentValue	:BYTE;
	(* message if the assertion is false *)
	message			:AssertMessage;
END_VAR
IF (NOT TO_BOOL(currentValue AND THIS^.LSB)) THEN
	THIS^.assertionWasWrong(message, THIS^.getDebugInfo('lsbIsSet'));
END_IF
END_METHOD

(*

## Short summary
This assertion method checks if the least significant bit of current value
is unset

.. <legal notes>

legal notes
=================
| SPDX-FileCopyrightText: © 2022 ekvip automation GmbH <info@ekvip.de>
| SPDX-License-Identifier: Apache-2.0
| For details check: Apache-2.0_

.. _Apache-2.0: https://www.apache.org/licenses/LICENSE-2.0

.. </legal notes>



*)

METHOD lsbIsUnset
VAR_INPUT
	(* current value to check *)
	currentValue	:BYTE;
	(* message if the assertion is false *)
	message			:AssertMessage;
END_VAR
IF (TO_BOOL(currentValue AND THIS^.LSB)) THEN
	THIS^.assertionWasWrong(message, THIS^.getDebugInfo('lsbIsUnset'));
END_IF
END_METHOD

(*

## Short summary
This assertion method checks if the most significant bit of current value
is equal to the expected value

.. <legal notes>

legal notes
=================
| SPDX-FileCopyrightText: © 2022 ekvip automation GmbH <info@ekvip.de>
| SPDX-License-Identifier: Apache-2.0
| For details check: Apache-2.0_

.. _Apache-2.0: https://www.apache.org/licenses/LICENSE-2.0

.. </legal notes>



*)

METHOD msbIsEqualTo
VAR_INPUT
	(* current value to check *)
	currentValue	:BYTE;
	(* expected value of msb *)
	expectedValue	:BOOL;
	(* message if the assertion is false *)
	message			:AssertMessage;
END_VAR
IF (TO_BOOL(currentValue AND THIS^.MSB) <> expectedValue) THEN
	THIS^.assertionWasWrong(message, THIS^.getDebugInfo('msbIsEqualTo'));
END_IF
END_METHOD

(*

## Short summary
This assertion method checks if the most significant bit of current value
is not equal to the unexpected value

.. <legal notes>

legal notes
=================
| SPDX-FileCopyrightText: © 2022 ekvip automation GmbH <info@ekvip.de>
| SPDX-License-Identifier: Apache-2.0
| For details check: Apache-2.0_

.. _Apache-2.0: https://www.apache.org/licenses/LICENSE-2.0

.. </legal notes>



*)

METHOD msbIsNotEqualTo
VAR_INPUT
	(* current value to check *)
	currentValue	:BYTE;
	(* unexpected value of msb *)
	unexpectedValue	:BOOL;
	(* message if the assertion is false *)
	message			:AssertMessage;
END_VAR
IF (TO_BOOL(currentValue AND THIS^.MSB) = unexpectedValue) THEN
	THIS^.assertionWasWrong(message, THIS^.getDebugInfo('msbIsNotEqualTo'));
END_IF
END_METHOD

(*

## Short summary
This assertion method checks if the most significant bit of current value
is set

.. <legal notes>

legal notes
=================
| SPDX-FileCopyrightText: © 2022 ekvip automation GmbH <info@ekvip.de>
| SPDX-License-Identifier: Apache-2.0
| For details check: Apache-2.0_

.. _Apache-2.0: https://www.apache.org/licenses/LICENSE-2.0

.. </legal notes>



*)

METHOD msbIsSet
VAR_INPUT
	(* current value to check *)
	currentValue	:BYTE;
	(* message if the assertion is false *)
	message			:AssertMessage;
END_VAR
IF (NOT TO_BOOL(currentValue AND THIS^.MSB)) THEN
	THIS^.assertionWasWrong(message, THIS^.getDebugInfo('msbIsSet'));
END_IF
END_METHOD

(*

## Short summary
This assertion method checks if the most significant bit of current value
is unset

.. <legal notes>

legal notes
=================
| SPDX-FileCopyrightText: © 2022 ekvip automation GmbH <info@ekvip.de>
| SPDX-License-Identifier: Apache-2.0
| For details check: Apache-2.0_

.. _Apache-2.0: https://www.apache.org/licenses/LICENSE-2.0

.. </legal notes>



*)

METHOD msbIsUnset
VAR_INPUT
	(* current value to check *)
	currentValue	:BYTE;
	(* message if the assertion is false *)
	message			:AssertMessage;
END_VAR
IF (TO_BOOL(currentValue AND THIS^.MSB)) THEN
	THIS^.assertionWasWrong(message, THIS^.getDebugInfo('msbIsUnset'));
END_IF
END_METHOD

(*

## Short summary
This assertion method checks if the result current value bitwise ``OR`` mask is equal to the expected value

.. <legal notes>

legal notes
=================
| SPDX-FileCopyrightText: © 2022 ekvip automation GmbH <info@ekvip.de>
| SPDX-License-Identifier: Apache-2.0
| For details check: Apache-2.0_

.. _Apache-2.0: https://www.apache.org/licenses/LICENSE-2.0

.. </legal notes>



*)

METHOD orMaskIsEqualTo
VAR_INPUT
	(* current value to check *)
	currentValue	:BYTE;
	(* 2nd operand for bitwise operation *)
	mask			:BYTE;
	(* expected result after masking *)
	expectedValue	:BYTE;
	(* message if the assertion is false *)
	message			:AssertMessage;
END_VAR
IF ((currentValue OR mask) <> expectedValue) THEN
	THIS^.assertionWasWrong(message, THIS^.getDebugInfo('orMaskIsEqualTo'));
END_IF
END_METHOD

(*

## Short summary
This assertion method checks if the result current value bitwise ``OR`` mask 
is not equal to the unexpected value

.. <legal notes>

legal notes
=================
| SPDX-FileCopyrightText: © 2022 ekvip automation GmbH <info@ekvip.de>
| SPDX-License-Identifier: Apache-2.0
| For details check: Apache-2.0_

.. _Apache-2.0: https://www.apache.org/licenses/LICENSE-2.0

.. </legal notes>



*)

METHOD orMaskIsNotEqualTo
VAR_INPUT
	(* current value to check *)
	currentValue	:BYTE;
	(* 2nd operand for bitwise operation *)
	mask			:BYTE;
	(* unexpected result after masking *)
	unexpectedValue	:BYTE;
	(* message if the assertion is false *)
	message			:AssertMessage;
END_VAR
IF ((currentValue OR mask) = unexpectedValue) THEN
	THIS^.assertionWasWrong(message, THIS^.getDebugInfo('orMaskIsNotEqualTo'));
END_IF
END_METHOD

(*

## Short summary
This assertion method checks if the current value is equal to the expected value

.. <legal notes>

legal notes
=================
| SPDX-FileCopyrightText: © 2022 ekvip automation GmbH <info@ekvip.de>
| SPDX-License-Identifier: Apache-2.0
| For details check: Apache-2.0_

.. _Apache-2.0: https://www.apache.org/licenses/LICENSE-2.0

.. </legal notes>



*)

METHOD valueIsEqualTo
VAR_INPUT
	(* current value to check *)
	currentValue	:BYTE;
	(* expected value to compare *)
	expectedValue	:BYTE;
	(* message if the assertion is false *)
	message			:AssertMessage;
END_VAR
IF (currentValue <> expectedValue) THEN
	THIS^.assertionWasWrong(message, THIS^.getDebugInfo('valueIsEqualTo'));
END_IF
END_METHOD

(*

## Short summary
This assertion method checks if the current value is greater than the less value

.. <legal notes>

legal notes
=================
| SPDX-FileCopyrightText: © 2022 ekvip automation GmbH <info@ekvip.de>
| SPDX-License-Identifier: Apache-2.0
| For details check: Apache-2.0_

.. _Apache-2.0: https://www.apache.org/licenses/LICENSE-2.0

.. </legal notes>



*)

METHOD valueIsGreaterThan
VAR_INPUT
	(* current value to check *)
	currentValue	:BYTE;
	(* less than lower limit *)
	lessValue		:BYTE;
	(* message if the assertion is false *)
	message			:AssertMessage;
END_VAR
IF (currentValue <= lessValue) THEN
	THIS^.assertionWasWrong(message, THIS^.getDebugInfo('valueIsGreaterThan'));
END_IF
END_METHOD

(*

## Short summary
This assertion method checks if the current value is inside a limit

**Attention:** 
	limits are included: ``valueIsInRangeOf(3, 3, 3)`` is a true assertion

.. <legal notes>

legal notes
=================
| SPDX-FileCopyrightText: © 2022 ekvip automation GmbH <info@ekvip.de>
| SPDX-License-Identifier: Apache-2.0
| For details check: Apache-2.0_

.. _Apache-2.0: https://www.apache.org/licenses/LICENSE-2.0

.. </legal notes>



*)

METHOD valueIsInRangeOf
VAR_INPUT
	(* lower limit for the current value *)
	lowerLimit		:BYTE;
	(* current value to check *)
	currentValue	:BYTE;
	(* upper limit for the current value *)
	upperLimit		:BYTE;
	(* message if the assertion is false *)
	message			:AssertMessage;
END_VAR
IF (
	(currentValue < lowerLimit)
	OR (currentValue > upperLimit)
) THEN
	THIS^.assertionWasWrong(message, THIS^.getDebugInfo('valueIsInRangeOf'));
END_IF
END_METHOD

(*

## Short summary
This assertion method checks if the current value is less than the greater value

.. <legal notes>

legal notes
=================
| SPDX-FileCopyrightText: © 2022 ekvip automation GmbH <info@ekvip.de>
| SPDX-License-Identifier: Apache-2.0
| For details check: Apache-2.0_

.. _Apache-2.0: https://www.apache.org/licenses/LICENSE-2.0

.. </legal notes>



*)

METHOD valueIsLessThan
VAR_INPUT
	(* current value to check *)
	currentValue	:BYTE;
	(* greater than upper limit *)
	greaterValue	:BYTE;
	(* message if the assertion is false *)
	message			:AssertMessage;
END_VAR
IF (currentValue >= greaterValue) THEN
	THIS^.assertionWasWrong(message, THIS^.getDebugInfo('valueIsLessThan'));
END_IF
END_METHOD

(*

## Short summary
This assertion method checks if the current value is less than or equal to the maximum value

.. <legal notes>

legal notes
=================
| SPDX-FileCopyrightText: © 2022 ekvip automation GmbH <info@ekvip.de>
| SPDX-License-Identifier: Apache-2.0
| For details check: Apache-2.0_

.. _Apache-2.0: https://www.apache.org/licenses/LICENSE-2.0

.. </legal notes>



*)

METHOD valueIsMax
VAR_INPUT
	(* current value to check *)
	currentValue	:BYTE;
	(* upper limit for the current value *)
	maximumValue	:BYTE;
	(* message if the assertion is false *)
	message			:AssertMessage;
END_VAR
IF (currentValue > maximumValue) THEN
	THIS^.assertionWasWrong(message, THIS^.getDebugInfo('valueIsMax'));
END_IF
END_METHOD

(*

## Short summary
This assertion method checks if the current value is greater than or equal to the minimum value

.. <legal notes>

legal notes
=================
| SPDX-FileCopyrightText: © 2022 ekvip automation GmbH <info@ekvip.de>
| SPDX-License-Identifier: Apache-2.0
| For details check: Apache-2.0_

.. _Apache-2.0: https://www.apache.org/licenses/LICENSE-2.0

.. </legal notes>



*)

METHOD valueIsMin
VAR_INPUT
	(* current value to check *)
	currentValue	:BYTE;
	(* lower limit for the current value *)
	minimumValue	:BYTE;
	(* message if the assertion is false *)
	message			:AssertMessage;
END_VAR
IF (currentValue < minimumValue) THEN
	THIS^.assertionWasWrong(message, THIS^.getDebugInfo('valueIsMin'));
END_IF
END_METHOD

(*

## Short summary
This assertion method checks if the current value is not equal to the unexpected value

.. <legal notes>

legal notes
=================
| SPDX-FileCopyrightText: © 2022 ekvip automation GmbH <info@ekvip.de>
| SPDX-License-Identifier: Apache-2.0
| For details check: Apache-2.0_

.. _Apache-2.0: https://www.apache.org/licenses/LICENSE-2.0

.. </legal notes>



*)

METHOD valueIsNotEqualTo
VAR_INPUT
	(* current value to check *)
	currentValue	:BYTE;
	(* unexpected value to compare *)
	unexpectedValue	:BYTE;
	(* message if the assertion is false *)
	message			:AssertMessage;
END_VAR
IF (currentValue = unexpectedValue) THEN
	THIS^.assertionWasWrong(message, THIS^.getDebugInfo('valueIsNotEqualTo'));
END_IF
END_METHOD

(*

## Short summary
This assertion method checks if the result current value bitwise ``XOR`` mask is equal to the expected value

.. <legal notes>

legal notes
=================
| SPDX-FileCopyrightText: © 2022 ekvip automation GmbH <info@ekvip.de>
| SPDX-License-Identifier: Apache-2.0
| For details check: Apache-2.0_

.. _Apache-2.0: https://www.apache.org/licenses/LICENSE-2.0

.. </legal notes>



*)

METHOD xorMaskIsEqualTo
VAR_INPUT
	(* current value to check *)
	currentValue	:BYTE;
	(* 2nd operand for bitwise operation *)
	mask			:BYTE;
	(* expected result after masking *)
	expectedValue	:BYTE;
	(* message if the assertion is false *)
	message			:AssertMessage;
END_VAR
IF ((currentValue XOR mask) <> expectedValue) THEN
	THIS^.assertionWasWrong(message, THIS^.getDebugInfo('xorMaskIsEqualTo'));
END_IF
END_METHOD

(*

## Short summary
This assertion method checks if the result current value bitwise ``XOR`` mask 
is not equal to the unexpected value

.. <legal notes>

legal notes
=================
| SPDX-FileCopyrightText: © 2022 ekvip automation GmbH <info@ekvip.de>
| SPDX-License-Identifier: Apache-2.0
| For details check: Apache-2.0_

.. _Apache-2.0: https://www.apache.org/licenses/LICENSE-2.0

.. </legal notes>



*)

METHOD xorMaskIsNotEqualTo
VAR_INPUT
	(* current value to check *)
	currentValue	:BYTE;
	(* 2nd operand for bitwise operation *)
	mask			:BYTE;
	(* unexpected result after masking *)
	unexpectedValue	:BYTE;
	(* message if the assertion is false *)
	message			:AssertMessage;
END_VAR
IF ((currentValue XOR mask) = unexpectedValue) THEN
	THIS^.assertionWasWrong(message, THIS^.getDebugInfo('xorMaskIsNotEqualTo'));
END_IF
END_METHOD

END_FUNCTION_BLOCK

// ---- Assertor/Assertions/BitNumberAssertions/classes/BitNumberAssertions.TcPOU
(*

## Short summary

 This class provides assert statements for bit numbers:
 It implements the interface `IBitNumberAssertions`
 For ``BYTE`` use `BitNumberAssertions.short`
 For ``WORD`` use `BitNumberAssertions.simple`
 For ``DWORD`` use `BitNumberAssertions.double`
 For ``LWORD`` use `BitNumberAssertions.long`
 For ``__XWORD`` use `BitNumberAssertions.x`

.. <legal notes>

legal notes
=================
| SPDX-FileCopyrightText: © 2022 ekvip automation GmbH <info@ekvip.de>
| SPDX-License-Identifier: Apache-2.0
| For details check: Apache-2.0_

.. _Apache-2.0: https://www.apache.org/licenses/LICENSE-2.0

.. </legal notes>



*)

{attribute 'reflection'}
FUNCTION_BLOCK INTERNAL BitNumberAssertions 
EXTENDS CNM_AbstractObject.Object 
IMPLEMENTS IBitNumberAssertions, IAssertCallBacksetter
VAR
	(* class to handle byte assertions *)
	byteAssertions	:ByteAssertions();
	(* class to handle word assertions *)
	wordAssertions	:WordAssertions();
	(* class to handle dword assertions *)
	dwordAssertions	:DWordAssertions();
	(* class to handle lword assertions *)
	lwordAssertions	:LWordAssertions();
	(* class to handle xword assertions *)
	xwordAssertions	:XWordAssertions();
END_VAR

(*

## Short summary
This abstract property returns the class name of the concrete object, 
It's for debugging purpose

.. <legal notes>

legal notes
=================
| SPDX-FileCopyrightText: © 2022 ekvip automation GmbH <info@ekvip.de>
| SPDX-License-Identifier: Apache-2.0
| For details check: Apache-2.0_

.. _Apache-2.0: https://www.apache.org/licenses/LICENSE-2.0

.. </legal notes>

*)

PROPERTY className :CNM_AbstractObject.ClassName
GET
className := 'CNM_Assertor.BitNumberAssertions';
END_GET
END_PROPERTY

(*

## Short summary
Returns the interface `IDwordAssertions`
with assert statements for double words ``DWORD`` 

.. <legal notes>

legal notes
=================
| SPDX-FileCopyrightText: © 2022 ekvip automation GmbH <info@ekvip.de>
| SPDX-License-Identifier: Apache-2.0
| For details check: Apache-2.0_

.. _Apache-2.0: https://www.apache.org/licenses/LICENSE-2.0

.. </legal notes>

*)

PROPERTY double :IDwordAssertions
GET
double := THIS^.dwordAssertions;
END_GET
END_PROPERTY

(*

## Short summary
Returns the interface `ILwordAssertions`
with assert statements for long words ``LWORD`` 

.. <legal notes>

legal notes
=================
| SPDX-FileCopyrightText: © 2022 ekvip automation GmbH <info@ekvip.de>
| SPDX-License-Identifier: Apache-2.0
| For details check: Apache-2.0_

.. _Apache-2.0: https://www.apache.org/licenses/LICENSE-2.0

.. </legal notes>

*)

PROPERTY long :ILwordAssertions
GET
long := THIS^.lwordAssertions;
END_GET
END_PROPERTY

(*

## Short summary
This methods is the setter for the callback class if an assertion was false

.. <legal notes>

legal notes
=================
| SPDX-FileCopyrightText: © 2022 ekvip automation GmbH <info@ekvip.de>
| SPDX-License-Identifier: Apache-2.0
| For details check: Apache-2.0_

.. _Apache-2.0: https://www.apache.org/licenses/LICENSE-2.0

.. </legal notes>



*)

METHOD setCallBack
VAR_INPUT
	(* the class that must be informed if an assertion is false *)
	callBack	:IAssertCallBack;  
END_VAR
THIS^.byteAssertions.setCallBack(callBack);
THIS^.wordAssertions.setCallBack(callBack);
THIS^.dwordAssertions.setCallBack(callBack);
THIS^.lwordAssertions.setCallBack(callBack);
THIS^.xwordAssertions.setCallBack(callBack);
END_METHOD

(*

## Short summary
Returns the interface `IByteAssertions`
with assert statements for bytes

.. <legal notes>

legal notes
=================
| SPDX-FileCopyrightText: © 2022 ekvip automation GmbH <info@ekvip.de>
| SPDX-License-Identifier: Apache-2.0
| For details check: Apache-2.0_

.. _Apache-2.0: https://www.apache.org/licenses/LICENSE-2.0

.. </legal notes>

*)

PROPERTY short :IByteAssertions
GET
short := THIS^.byteAssertions;
END_GET
END_PROPERTY

(*

## Short summary
Returns the interface `IWordAssertions`
with assert statements for words 

.. <legal notes>

legal notes
=================
| SPDX-FileCopyrightText: © 2022 ekvip automation GmbH <info@ekvip.de>
| SPDX-License-Identifier: Apache-2.0
| For details check: Apache-2.0_

.. _Apache-2.0: https://www.apache.org/licenses/LICENSE-2.0

.. </legal notes>

*)

PROPERTY simple :IWordAssertions
GET
simple := THIS^.wordAssertions;
END_GET
END_PROPERTY

(*

## Short summary
Returns the interface `IXwordAssertions`
with assert statements for register length words ``__XWORD``

.. <legal notes>

legal notes
=================
| SPDX-FileCopyrightText: © 2022 ekvip automation GmbH <info@ekvip.de>
| SPDX-License-Identifier: Apache-2.0
| For details check: Apache-2.0_

.. _Apache-2.0: https://www.apache.org/licenses/LICENSE-2.0

.. </legal notes>

*)

PROPERTY x :IXwordAssertions
GET
x := THIS^.xwordAssertions;
END_GET
END_PROPERTY

END_FUNCTION_BLOCK

// ---- Assertor/Assertions/BitNumberAssertions/Word/classes/WordAssertions.TcPOU
(*

## Short summary
This class provides assert statements for words  

.. <legal notes>

legal notes
=================
| SPDX-FileCopyrightText: © 2022 ekvip automation GmbH <info@ekvip.de>
| SPDX-License-Identifier: Apache-2.0
| For details check: Apache-2.0_

.. _Apache-2.0: https://www.apache.org/licenses/LICENSE-2.0

.. </legal notes>



*)

{attribute 'reflection'}
FUNCTION_BLOCK INTERNAL WordAssertions EXTENDS AbstractAssertion IMPLEMENTS IWordAssertions
VAR
END_VAR
VAR CONSTANT
	(* least significant bit *)
	LSB	:WORD := 16#0001;
	(* most significant bit *)
	MSB :WORD := 16#8000;
END_VAR

(*

## Short summary
This assertion method checks if the result current value bitwise ``AND`` mask is equal to the expected value

.. <legal notes>

legal notes
=================
| SPDX-FileCopyrightText: © 2022 ekvip automation GmbH <info@ekvip.de>
| SPDX-License-Identifier: Apache-2.0
| For details check: Apache-2.0_

.. _Apache-2.0: https://www.apache.org/licenses/LICENSE-2.0

.. </legal notes>



*)

METHOD andMaskIsEqualTo
VAR_INPUT
	(* current value to check *)
	currentValue	:WORD;
	(* 2nd operand for bitwise operation *)
	mask			:WORD;
	(* expected result after masking *)
	expectedValue	:WORD;
	(* message if the assertion is false *)
	message			:AssertMessage;
END_VAR
IF ((currentValue AND mask) <> expectedValue) THEN
	THIS^.assertionWasWrong(message, THIS^.getDebugInfo('andMaskIsEqualTo'));
END_IF
END_METHOD

(*

## Short summary
This assertion method checks if the result current value bitwise ``AND`` mask
is not equal to the unexpected value

.. <legal notes>

legal notes
=================
| SPDX-FileCopyrightText: © 2022 ekvip automation GmbH <info@ekvip.de>
| SPDX-License-Identifier: Apache-2.0
| For details check: Apache-2.0_

.. _Apache-2.0: https://www.apache.org/licenses/LICENSE-2.0

.. </legal notes>



*)

METHOD andMaskIsNotEqualTo
VAR_INPUT
	(* current value to check *)
	currentValue	:WORD;
	(* 2nd operand for bitwise operation *)
	mask			:WORD;
	(* unexpected result after masking *)
	unexpectedValue	:WORD;
	(* message if the assertion is false *)
	message			:AssertMessage;
END_VAR
IF ((currentValue AND mask) = unexpectedValue) THEN
	THIS^.assertionWasWrong(message, THIS^.getDebugInfo('andMaskIsNotEqualTo'));
END_IF
END_METHOD

(*

## Short summary
This assertion method checks if the selected bit of current value
is equal to the expected value

.. <legal notes>

legal notes
=================
| SPDX-FileCopyrightText: © 2022 ekvip automation GmbH <info@ekvip.de>
| SPDX-License-Identifier: Apache-2.0
| For details check: Apache-2.0_

.. _Apache-2.0: https://www.apache.org/licenses/LICENSE-2.0

.. </legal notes>



*)

METHOD bitXIsEqualTo
VAR_INPUT
	(* current value to check *)
	currentValue	:WORD;
	(* number of bit to check *)
	number			:BitNumberWord;
	(* expected value of bit *)
	expectedValue	:BOOL;
	(* message if the assertion is false *)
	message			:AssertMessage;
END_VAR
IF (
	TO_BOOL(
		TO_WORD(SHL(THIS^.LSB, number))
		AND currentValue
	) <> expectedValue
) THEN
	THIS^.assertionWasWrong(message, THIS^.getDebugInfo('bitXIsEqualTo'));
END_IF
END_METHOD

(*

## Short summary
This assertion method checks if the selected bit of current value
is not equal to the unexpected value

.. <legal notes>

legal notes
=================
| SPDX-FileCopyrightText: © 2022 ekvip automation GmbH <info@ekvip.de>
| SPDX-License-Identifier: Apache-2.0
| For details check: Apache-2.0_

.. _Apache-2.0: https://www.apache.org/licenses/LICENSE-2.0

.. </legal notes>



*)

METHOD bitXIsNotEqualTo
VAR_INPUT
	(* current value to check *)
	currentValue	:WORD;
	(* number of bit to check *)
	number			:BitNumberWord;
	(* unexpected value of bit *)
	unexpectedValue	:BOOL;
	(* message if the assertion is false *)
	message			:AssertMessage;
END_VAR
IF (
	TO_BOOL(
		TO_WORD(SHL(THIS^.LSB, number))
		AND currentValue
	) = unexpectedValue
) THEN
	THIS^.assertionWasWrong(message, THIS^.getDebugInfo('bitXIsNotEqualTo'));
END_IF
END_METHOD

(*

## Short summary
This assertion method checks if the selected bit of current value
is set

.. <legal notes>

legal notes
=================
| SPDX-FileCopyrightText: © 2022 ekvip automation GmbH <info@ekvip.de>
| SPDX-License-Identifier: Apache-2.0
| For details check: Apache-2.0_

.. _Apache-2.0: https://www.apache.org/licenses/LICENSE-2.0

.. </legal notes>



*)

METHOD bitXIsSet
VAR_INPUT
	(* current value to check *)
	currentValue	:WORD;
	(* number of bit to check *)
	number			:BitNumberWord;
	(* message if the assertion is false *)
	message			:AssertMessage;
END_VAR
IF (
	NOT TO_BOOL(
		TO_WORD(SHL(THIS^.LSB, number))
		AND currentValue
	)
) THEN
	THIS^.assertionWasWrong(message, THIS^.getDebugInfo('bitXIsSet'));
END_IF
END_METHOD

(*

## Short summary
This assertion method checks if the selected bit of current value
is unset

.. <legal notes>

legal notes
=================
| SPDX-FileCopyrightText: © 2022 ekvip automation GmbH <info@ekvip.de>
| SPDX-License-Identifier: Apache-2.0
| For details check: Apache-2.0_

.. _Apache-2.0: https://www.apache.org/licenses/LICENSE-2.0

.. </legal notes>



*)

METHOD bitXIsUnset
VAR_INPUT
	(* current value to check *)
	currentValue	:WORD;
	(* number of bit to check *)
	number			:BitNumberWord;
	(* message if the assertion is false *)
	message			:AssertMessage;
END_VAR
IF (
	TO_BOOL(
		TO_WORD(SHL(THIS^.LSB, number))
		AND currentValue
	)
) THEN
	THIS^.assertionWasWrong(message, THIS^.getDebugInfo('bitXIsUnset'));
END_IF
END_METHOD

(*

## Short summary
This abstract property returns the class name of the concrete object, 
It's for debugging purpose

.. <legal notes>

legal notes
=================
| SPDX-FileCopyrightText: © 2022 ekvip automation GmbH <info@ekvip.de>
| SPDX-License-Identifier: Apache-2.0
| For details check: Apache-2.0_

.. _Apache-2.0: https://www.apache.org/licenses/LICENSE-2.0

.. </legal notes>

*)

PROPERTY className :CNM_AbstractObject.ClassName
GET
className := 'CNM_Assertor.WordAssertions';
END_GET
END_PROPERTY

(*

## Short summary
This assertion method checks if the least significant bit of current value
is equal to the expected value

.. <legal notes>

legal notes
=================
| SPDX-FileCopyrightText: © 2022 ekvip automation GmbH <info@ekvip.de>
| SPDX-License-Identifier: Apache-2.0
| For details check: Apache-2.0_

.. _Apache-2.0: https://www.apache.org/licenses/LICENSE-2.0

.. </legal notes>



*)

METHOD lsbIsEqualTo
VAR_INPUT
	(* current value to check *)
	currentValue	:WORD;
	(* expected value of lsb *)
	expectedValue	:BOOL;
	(* message if the assertion is false *)
	message			:AssertMessage;
END_VAR
IF (TO_BOOL(currentValue AND THIS^.LSB) <> expectedValue) THEN
	THIS^.assertionWasWrong(message, THIS^.getDebugInfo('lsbIsEqualTo'));
END_IF
END_METHOD

(*

## Short summary
This assertion method checks if the least significant bit of current value
is not equal to the unexpected value

.. <legal notes>

legal notes
=================
| SPDX-FileCopyrightText: © 2022 ekvip automation GmbH <info@ekvip.de>
| SPDX-License-Identifier: Apache-2.0
| For details check: Apache-2.0_

.. _Apache-2.0: https://www.apache.org/licenses/LICENSE-2.0

.. </legal notes>



*)

METHOD lsbIsNotEqualTo
VAR_INPUT
	(* current value to check *)
	currentValue	:WORD;
	(* unexpected value of lsb *)
	unexpectedValue	:BOOL;
	(* message if the assertion is false *)
	message			:AssertMessage;
END_VAR
IF (TO_BOOL(currentValue AND THIS^.LSB) = unexpectedValue) THEN
	THIS^.assertionWasWrong(message, THIS^.getDebugInfo('lsbIsNotEqualTo'));
END_IF
END_METHOD

(*

## Short summary
This assertion method checks if the least significant bit of current value
is set

.. <legal notes>

legal notes
=================
| SPDX-FileCopyrightText: © 2022 ekvip automation GmbH <info@ekvip.de>
| SPDX-License-Identifier: Apache-2.0
| For details check: Apache-2.0_

.. _Apache-2.0: https://www.apache.org/licenses/LICENSE-2.0

.. </legal notes>



*)

METHOD lsbIsSet
VAR_INPUT
	(* current value to check *)
	currentValue	:WORD;
	(* message if the assertion is false *)
	message			:AssertMessage;
END_VAR
IF (NOT TO_BOOL(currentValue AND THIS^.LSB)) THEN
	THIS^.assertionWasWrong(message, THIS^.getDebugInfo('lsbIsSet'));
END_IF
END_METHOD

(*

## Short summary
This assertion method checks if the least significant bit of current value
is unset

.. <legal notes>

legal notes
=================
| SPDX-FileCopyrightText: © 2022 ekvip automation GmbH <info@ekvip.de>
| SPDX-License-Identifier: Apache-2.0
| For details check: Apache-2.0_

.. _Apache-2.0: https://www.apache.org/licenses/LICENSE-2.0

.. </legal notes>



*)

METHOD lsbIsUnset
VAR_INPUT
	(* current value to check *)
	currentValue	:WORD;
	(* message if the assertion is false *)
	message			:AssertMessage;
END_VAR
IF (TO_BOOL(currentValue AND THIS^.LSB)) THEN
	THIS^.assertionWasWrong(message, THIS^.getDebugInfo('lsbIsUnset'));
END_IF
END_METHOD

(*

## Short summary
This assertion method checks if the most significant bit of current value
is equal to the expected value

.. <legal notes>

legal notes
=================
| SPDX-FileCopyrightText: © 2022 ekvip automation GmbH <info@ekvip.de>
| SPDX-License-Identifier: Apache-2.0
| For details check: Apache-2.0_

.. _Apache-2.0: https://www.apache.org/licenses/LICENSE-2.0

.. </legal notes>



*)

METHOD msbIsEqualTo
VAR_INPUT
	(* current value to check *)
	currentValue	:WORD;
	(* expected value of msb *)
	expectedValue	:BOOL;
	(* message if the assertion is false *)
	message			:AssertMessage;
END_VAR
IF (TO_BOOL(currentValue AND THIS^.MSB) <> expectedValue) THEN
	THIS^.assertionWasWrong(message, THIS^.getDebugInfo('msbIsEqualTo'));
END_IF
END_METHOD

(*

## Short summary
This assertion method checks if the most significant bit of current value
is not equal to the unexpected value

.. <legal notes>

legal notes
=================
| SPDX-FileCopyrightText: © 2022 ekvip automation GmbH <info@ekvip.de>
| SPDX-License-Identifier: Apache-2.0
| For details check: Apache-2.0_

.. _Apache-2.0: https://www.apache.org/licenses/LICENSE-2.0

.. </legal notes>



*)

METHOD msbIsNotEqualTo
VAR_INPUT
	(* current value to check *)
	currentValue	:WORD;
	(* unexpected value of msb *)
	unexpectedValue	:BOOL;
	(* message if the assertion is false *)
	message			:AssertMessage;
END_VAR
IF (TO_BOOL(currentValue AND THIS^.MSB) = unexpectedValue) THEN
	THIS^.assertionWasWrong(message, THIS^.getDebugInfo('msbIsNotEqualTo'));
END_IF
END_METHOD

(*

## Short summary
This assertion method checks if the most significant bit of current value
is set

.. <legal notes>

legal notes
=================
| SPDX-FileCopyrightText: © 2022 ekvip automation GmbH <info@ekvip.de>
| SPDX-License-Identifier: Apache-2.0
| For details check: Apache-2.0_

.. _Apache-2.0: https://www.apache.org/licenses/LICENSE-2.0

.. </legal notes>



*)

METHOD msbIsSet
VAR_INPUT
	(* current value to check *)
	currentValue	:WORD;
	(* message if the assertion is false *)
	message			:AssertMessage;
END_VAR
IF (NOT TO_BOOL(currentValue AND THIS^.MSB)) THEN
	THIS^.assertionWasWrong(message, THIS^.getDebugInfo('msbIsSet'));
END_IF
END_METHOD

(*

## Short summary
This assertion method checks if the most significant bit of current value
is unset

.. <legal notes>

legal notes
=================
| SPDX-FileCopyrightText: © 2022 ekvip automation GmbH <info@ekvip.de>
| SPDX-License-Identifier: Apache-2.0
| For details check: Apache-2.0_

.. _Apache-2.0: https://www.apache.org/licenses/LICENSE-2.0

.. </legal notes>



*)

METHOD msbIsUnset
VAR_INPUT
	(* current value to check *)
	currentValue	:WORD;
	(* message if the assertion is false *)
	message			:AssertMessage;
END_VAR
IF (TO_BOOL(currentValue AND THIS^.MSB)) THEN
	THIS^.assertionWasWrong(message, THIS^.getDebugInfo('msbIsUnset'));
END_IF
END_METHOD

(*

## Short summary
This assertion method checks if the result current value bitwise ``OR`` mask is equal to the expected value

.. <legal notes>

legal notes
=================
| SPDX-FileCopyrightText: © 2022 ekvip automation GmbH <info@ekvip.de>
| SPDX-License-Identifier: Apache-2.0
| For details check: Apache-2.0_

.. _Apache-2.0: https://www.apache.org/licenses/LICENSE-2.0

.. </legal notes>



*)

METHOD orMaskIsEqualTo
VAR_INPUT
	(* current value to check *)
	currentValue	:WORD;
	(* 2nd operand for bitwise operation *)
	mask			:WORD;
	(* expected result after masking *)
	expectedValue	:WORD;
	(* message if the assertion is false *)
	message			:AssertMessage;
END_VAR
IF ((currentValue OR mask) <> expectedValue) THEN
	THIS^.assertionWasWrong(message, THIS^.getDebugInfo('orMaskIsEqualTo'));
END_IF
END_METHOD

(*

## Short summary
This assertion method checks if the result current value bitwise ``OR`` mask 
is not equal to the unexpected value

.. <legal notes>

legal notes
=================
| SPDX-FileCopyrightText: © 2022 ekvip automation GmbH <info@ekvip.de>
| SPDX-License-Identifier: Apache-2.0
| For details check: Apache-2.0_

.. _Apache-2.0: https://www.apache.org/licenses/LICENSE-2.0

.. </legal notes>



*)

METHOD orMaskIsNotEqualTo
VAR_INPUT
	(* current value to check *)
	currentValue	:WORD;
	(* 2nd operand for bitwise operation *)
	mask			:WORD;
	(* unexpected result after masking *)
	unexpectedValue	:WORD;
	(* message if the assertion is false *)
	message			:AssertMessage;
END_VAR
IF ((currentValue OR mask) = unexpectedValue) THEN
	THIS^.assertionWasWrong(message, THIS^.getDebugInfo('orMaskIsNotEqualTo'));
END_IF
END_METHOD

(*

## Short summary
This assertion method checks if the current value is equal to the expected value

.. <legal notes>

legal notes
=================
| SPDX-FileCopyrightText: © 2022 ekvip automation GmbH <info@ekvip.de>
| SPDX-License-Identifier: Apache-2.0
| For details check: Apache-2.0_

.. _Apache-2.0: https://www.apache.org/licenses/LICENSE-2.0

.. </legal notes>



*)

METHOD valueIsEqualTo
VAR_INPUT
	(* current value to check *)
	currentValue	:WORD;
	(* expected value to compare *)
	expectedValue	:WORD;
	(* message if the assertion is false *)
	message			:AssertMessage;
END_VAR
IF (currentValue <> expectedValue) THEN
	THIS^.assertionWasWrong(message, THIS^.getDebugInfo('valueIsEqualTo'));
END_IF
END_METHOD

(*

## Short summary
This assertion method checks if the current value is greater than the less value

.. <legal notes>

legal notes
=================
| SPDX-FileCopyrightText: © 2022 ekvip automation GmbH <info@ekvip.de>
| SPDX-License-Identifier: Apache-2.0
| For details check: Apache-2.0_

.. _Apache-2.0: https://www.apache.org/licenses/LICENSE-2.0

.. </legal notes>



*)

METHOD valueIsGreaterThan
VAR_INPUT
	(* current value to check *)
	currentValue	:WORD;
	(* less than lower limit *)
	lessValue		:WORD;
	(* message if the assertion is false *)
	message			:AssertMessage;
END_VAR
IF (currentValue <= lessValue) THEN
	THIS^.assertionWasWrong(message, THIS^.getDebugInfo('valueIsGreaterThan'));
END_IF
END_METHOD

(*

## Short summary
This assertion method checks if the current value is inside a limit

**Attention:** 
	limits are included: ``valueIsInRangeOf(3, 3, 3)`` is a true assertion

.. <legal notes>

legal notes
=================
| SPDX-FileCopyrightText: © 2022 ekvip automation GmbH <info@ekvip.de>
| SPDX-License-Identifier: Apache-2.0
| For details check: Apache-2.0_

.. _Apache-2.0: https://www.apache.org/licenses/LICENSE-2.0

.. </legal notes>



*)

METHOD valueIsInRangeOf
VAR_INPUT
	(* lower limit for the current value *)
	lowerLimit		:WORD;
	(* current value to check *)
	currentValue	:WORD;
	(* upper limit for the current value *)
	upperLimit		:WORD;
	(* message if the assertion is false *)
	message			:AssertMessage;
END_VAR
IF (
	(currentValue < lowerLimit)
	OR (currentValue > upperLimit)
) THEN
	THIS^.assertionWasWrong(message, THIS^.getDebugInfo('valueIsInRangeOf'));
END_IF
END_METHOD

(*

## Short summary
This assertion method checks if the current value is less than the greater value

.. <legal notes>

legal notes
=================
| SPDX-FileCopyrightText: © 2022 ekvip automation GmbH <info@ekvip.de>
| SPDX-License-Identifier: Apache-2.0
| For details check: Apache-2.0_

.. _Apache-2.0: https://www.apache.org/licenses/LICENSE-2.0

.. </legal notes>



*)

METHOD valueIsLessThan
VAR_INPUT
	(* current value to check *)
	currentValue	:WORD;
	(* greater than upper limit *)
	greaterValue	:WORD;
	(* message if the assertion is false *)
	message			:AssertMessage;
END_VAR
IF (currentValue >= greaterValue) THEN
	THIS^.assertionWasWrong(message, THIS^.getDebugInfo('valueIsLessThan'));
END_IF
END_METHOD

(*

## Short summary
This assertion method checks if the current value is less than or equal to the maximum value

.. <legal notes>

legal notes
=================
| SPDX-FileCopyrightText: © 2022 ekvip automation GmbH <info@ekvip.de>
| SPDX-License-Identifier: Apache-2.0
| For details check: Apache-2.0_

.. _Apache-2.0: https://www.apache.org/licenses/LICENSE-2.0

.. </legal notes>



*)

METHOD valueIsMax
VAR_INPUT
	(* current value to check *)
	currentValue	:WORD;
	(* upper limit for the current value *)
	maximumValue	:WORD;
	(* message if the assertion is false *)
	message			:AssertMessage;
END_VAR
IF (currentValue > maximumValue) THEN
	THIS^.assertionWasWrong(message, THIS^.getDebugInfo('valueIsMax'));
END_IF
END_METHOD

(*

## Short summary
This assertion method checks if the current value is greater than or equal to the minimum value

.. <legal notes>

legal notes
=================
| SPDX-FileCopyrightText: © 2022 ekvip automation GmbH <info@ekvip.de>
| SPDX-License-Identifier: Apache-2.0
| For details check: Apache-2.0_

.. _Apache-2.0: https://www.apache.org/licenses/LICENSE-2.0

.. </legal notes>



*)

METHOD valueIsMin
VAR_INPUT
	(* current value to check *)
	currentValue	:WORD;
	(* lower limit for the current value *)
	minimumValue	:WORD;
	(* message if the assertion is false *)
	message			:AssertMessage;
END_VAR
IF (currentValue < minimumValue) THEN
	THIS^.assertionWasWrong(message, THIS^.getDebugInfo('valueIsMin'));
END_IF
END_METHOD

(*

## Short summary
This assertion method checks if the current value is not equal to the unexpected value

.. <legal notes>

legal notes
=================
| SPDX-FileCopyrightText: © 2022 ekvip automation GmbH <info@ekvip.de>
| SPDX-License-Identifier: Apache-2.0
| For details check: Apache-2.0_

.. _Apache-2.0: https://www.apache.org/licenses/LICENSE-2.0

.. </legal notes>



*)

METHOD valueIsNotEqualTo
VAR_INPUT
	(* current value to check *)
	currentValue	:WORD;
	(* unexpected value to compare *)
	unexpectedValue	:WORD;
	(* message if the assertion is false *)
	message			:AssertMessage;
END_VAR
IF (currentValue = unexpectedValue) THEN
	THIS^.assertionWasWrong(message, THIS^.getDebugInfo('valueIsNotEqualTo'));
END_IF
END_METHOD

(*

## Short summary
This assertion method checks if the result current value bitwise ``XOR`` mask is equal to the expected value

.. <legal notes>

legal notes
=================
| SPDX-FileCopyrightText: © 2022 ekvip automation GmbH <info@ekvip.de>
| SPDX-License-Identifier: Apache-2.0
| For details check: Apache-2.0_

.. _Apache-2.0: https://www.apache.org/licenses/LICENSE-2.0

.. </legal notes>



*)

METHOD xorMaskIsEqualTo
VAR_INPUT
	(* current value to check *)
	currentValue	:WORD;
	(* 2nd operand for bitwise operation *)
	mask			:WORD;
	(* expected result after masking *)
	expectedValue	:WORD;
	(* message if the assertion is false *)
	message			:AssertMessage;
END_VAR
IF ((currentValue XOR mask) <> expectedValue) THEN
	THIS^.assertionWasWrong(message, THIS^.getDebugInfo('xorMaskIsEqualTo'));
END_IF
END_METHOD

(*

## Short summary
This assertion method checks if the result current value bitwise ``XOR`` mask 
is not equal to the unexpected value

.. <legal notes>

legal notes
=================
| SPDX-FileCopyrightText: © 2022 ekvip automation GmbH <info@ekvip.de>
| SPDX-License-Identifier: Apache-2.0
| For details check: Apache-2.0_

.. _Apache-2.0: https://www.apache.org/licenses/LICENSE-2.0

.. </legal notes>



*)

METHOD xorMaskIsNotEqualTo
VAR_INPUT
	(* current value to check *)
	currentValue	:WORD;
	(* 2nd operand for bitwise operation *)
	mask			:WORD;
	(* unexpected result after masking *)
	unexpectedValue	:WORD;
	(* message if the assertion is false *)
	message			:AssertMessage;
END_VAR
IF ((currentValue XOR mask) = unexpectedValue) THEN
	THIS^.assertionWasWrong(message, THIS^.getDebugInfo('xorMaskIsNotEqualTo'));
END_IF
END_METHOD

END_FUNCTION_BLOCK

// ---- Assertor/Assertions/BitNumberAssertions/Dword/classes/DWordAssertions.TcPOU
(*

## Short summary
This class provides assert statements for double words 

.. <legal notes>

legal notes
=================
| SPDX-FileCopyrightText: © 2022 ekvip automation GmbH <info@ekvip.de>
| SPDX-License-Identifier: Apache-2.0
| For details check: Apache-2.0_

.. _Apache-2.0: https://www.apache.org/licenses/LICENSE-2.0

.. </legal notes>



*)

{attribute 'reflection'}
FUNCTION_BLOCK INTERNAL DWordAssertions EXTENDS AbstractAssertion IMPLEMENTS IDWordAssertions
VAR
END_VAR
VAR CONSTANT
	(* least significant bit *)
	LSB	:DWORD := 16#0000_0001;
	(* most significant bit *)
	MSB :DWORD := 16#8000_0000;
END_VAR

(*

## Short summary
This assertion method checks if the result current value bitwise ``AND`` mask is equal to the expected value

.. <legal notes>

legal notes
=================
| SPDX-FileCopyrightText: © 2022 ekvip automation GmbH <info@ekvip.de>
| SPDX-License-Identifier: Apache-2.0
| For details check: Apache-2.0_

.. _Apache-2.0: https://www.apache.org/licenses/LICENSE-2.0

.. </legal notes>



*)

METHOD andMaskIsEqualTo
VAR_INPUT
	(* current value to check *)
	currentValue	:DWORD;
	(* 2nd operand for bitwise operation *)
	mask			:DWORD;
	(* expected result after masking *)
	expectedValue	:DWORD;
	(* message if the assertion is false *)
	message			:AssertMessage;
END_VAR
IF ((currentValue AND mask) <> expectedValue) THEN
	THIS^.assertionWasWrong(message, THIS^.getDebugInfo('andMaskIsEqualTo'));
END_IF
END_METHOD

(*

## Short summary
This assertion method checks if the result current value bitwise ``AND`` mask
is not equal to the unexpected value

.. <legal notes>

legal notes
=================
| SPDX-FileCopyrightText: © 2022 ekvip automation GmbH <info@ekvip.de>
| SPDX-License-Identifier: Apache-2.0
| For details check: Apache-2.0_

.. _Apache-2.0: https://www.apache.org/licenses/LICENSE-2.0

.. </legal notes>



*)

METHOD andMaskIsNotEqualTo
VAR_INPUT
	(* current value to check *)
	currentValue	:DWORD;
	(* 2nd operand for bitwise operation *)
	mask			:DWORD;
	(* unexpected result after masking *)
	unexpectedValue	:DWORD;
	(* message if the assertion is false *)
	message			:AssertMessage;
END_VAR
IF ((currentValue AND mask) = unexpectedValue) THEN
	THIS^.assertionWasWrong(message, THIS^.getDebugInfo('andMaskIsNotEqualTo'));
END_IF
END_METHOD

(*

## Short summary
This assertion method checks if the selected bit of current value
is equal to the expected value

.. <legal notes>

legal notes
=================
| SPDX-FileCopyrightText: © 2022 ekvip automation GmbH <info@ekvip.de>
| SPDX-License-Identifier: Apache-2.0
| For details check: Apache-2.0_

.. _Apache-2.0: https://www.apache.org/licenses/LICENSE-2.0

.. </legal notes>



*)

METHOD bitXIsEqualTo
VAR_INPUT
	(* current value to check *)
	currentValue	:DWORD;
	(* number of bit to check *)
	number			:BitNumberDWord;
	(* expected value of bit *)
	expectedValue	:BOOL;
	(* message if the assertion is false *)
	message			:AssertMessage;
END_VAR
IF (
	TO_BOOL(
		TO_DWORD(SHL(THIS^.LSB, number))
		AND currentValue
	) <> expectedValue
) THEN
	THIS^.assertionWasWrong(message, THIS^.getDebugInfo('bitXIsEqualTo'));
END_IF
END_METHOD

(*

## Short summary
This assertion method checks if the selected bit of current value
is not equal to the unexpected value

.. <legal notes>

legal notes
=================
| SPDX-FileCopyrightText: © 2022 ekvip automation GmbH <info@ekvip.de>
| SPDX-License-Identifier: Apache-2.0
| For details check: Apache-2.0_

.. _Apache-2.0: https://www.apache.org/licenses/LICENSE-2.0

.. </legal notes>



*)

METHOD bitXIsNotEqualTo
VAR_INPUT
	(* current value to check *)
	currentValue	:DWORD;
	(* number of bit to check *)
	number			:BitNumberDWord;
	(* unexpected value of bit *)
	unexpectedValue	:BOOL;
	(* message if the assertion is false *)
	message			:AssertMessage;
END_VAR
IF (
	TO_BOOL(
		TO_DWORD(SHL(THIS^.LSB, number))
		AND currentValue
	) = unexpectedValue
) THEN
	THIS^.assertionWasWrong(message, THIS^.getDebugInfo('bitXIsNotEqualTo'));
END_IF
END_METHOD

(*

## Short summary
This assertion method checks if the selected bit of current value
is set

.. <legal notes>

legal notes
=================
| SPDX-FileCopyrightText: © 2022 ekvip automation GmbH <info@ekvip.de>
| SPDX-License-Identifier: Apache-2.0
| For details check: Apache-2.0_

.. _Apache-2.0: https://www.apache.org/licenses/LICENSE-2.0

.. </legal notes>



*)

METHOD bitXIsSet
VAR_INPUT
	(* current value to check *)
	currentValue	:DWORD;
	(* number of bit to check *)
	number			:BitNumberDWord;
	(* message if the assertion is false *)
	message			:AssertMessage;
END_VAR
IF (
	NOT TO_BOOL(
		TO_DWORD(SHL(THIS^.LSB, number))
		AND currentValue
	)
) THEN
	THIS^.assertionWasWrong(message, THIS^.getDebugInfo('bitXIsSet'));
END_IF
END_METHOD

(*

## Short summary
This assertion method checks if the selected bit of current value
is unset

.. <legal notes>

legal notes
=================
| SPDX-FileCopyrightText: © 2022 ekvip automation GmbH <info@ekvip.de>
| SPDX-License-Identifier: Apache-2.0
| For details check: Apache-2.0_

.. _Apache-2.0: https://www.apache.org/licenses/LICENSE-2.0

.. </legal notes>



*)

METHOD bitXIsUnset
VAR_INPUT
	(* current value to check *)
	currentValue	:DWORD;
	(* number of bit to check *)
	number			:BitNumberDWord;
	(* message if the assertion is false *)
	message			:AssertMessage;
END_VAR
IF (
	TO_BOOL(
		TO_DWORD(SHL(THIS^.LSB, number))
		AND currentValue
	)
) THEN
	THIS^.assertionWasWrong(message, THIS^.getDebugInfo('bitXIsUnset'));
END_IF
END_METHOD

(*

## Short summary
This abstract property returns the class name of the concrete object, 
It's for debugging purpose

.. <legal notes>

legal notes
=================
| SPDX-FileCopyrightText: © 2022 ekvip automation GmbH <info@ekvip.de>
| SPDX-License-Identifier: Apache-2.0
| For details check: Apache-2.0_

.. _Apache-2.0: https://www.apache.org/licenses/LICENSE-2.0

.. </legal notes>

*)

PROPERTY className :CNM_AbstractObject.ClassName
GET
className := 'CNM_Assertor.DWordAssertions';
END_GET
END_PROPERTY

(*

## Short summary
This assertion method checks if the least significant bit of current value
is equal to the expected value

.. <legal notes>

legal notes
=================
| SPDX-FileCopyrightText: © 2022 ekvip automation GmbH <info@ekvip.de>
| SPDX-License-Identifier: Apache-2.0
| For details check: Apache-2.0_

.. _Apache-2.0: https://www.apache.org/licenses/LICENSE-2.0

.. </legal notes>



*)

METHOD lsbIsEqualTo
VAR_INPUT
	(* current value to check *)
	currentValue	:DWORD;
	(* expected value of lsb *)
	expectedValue	:BOOL;
	(* message if the assertion is false *)
	message			:AssertMessage;
END_VAR
IF (TO_BOOL(currentValue AND THIS^.LSB) <> expectedValue) THEN
	THIS^.assertionWasWrong(message, THIS^.getDebugInfo('lsbIsEqualTo'));
END_IF
END_METHOD

(*

## Short summary
This assertion method checks if the least significant bit of current value
is not equal to the unexpected value

.. <legal notes>

legal notes
=================
| SPDX-FileCopyrightText: © 2022 ekvip automation GmbH <info@ekvip.de>
| SPDX-License-Identifier: Apache-2.0
| For details check: Apache-2.0_

.. _Apache-2.0: https://www.apache.org/licenses/LICENSE-2.0

.. </legal notes>



*)

METHOD lsbIsNotEqualTo
VAR_INPUT
	(* current value to check *)
	currentValue	:DWORD;
	(* unexpected value of lsb *)
	unexpectedValue	:BOOL;
	(* message if the assertion is false *)
	message			:AssertMessage;
END_VAR
IF (TO_BOOL(currentValue AND THIS^.LSB) = unexpectedValue) THEN
	THIS^.assertionWasWrong(message, THIS^.getDebugInfo('lsbIsNotEqualTo'));
END_IF
END_METHOD

(*

## Short summary
This assertion method checks if the least significant bit of current value
is set

.. <legal notes>

legal notes
=================
| SPDX-FileCopyrightText: © 2022 ekvip automation GmbH <info@ekvip.de>
| SPDX-License-Identifier: Apache-2.0
| For details check: Apache-2.0_

.. _Apache-2.0: https://www.apache.org/licenses/LICENSE-2.0

.. </legal notes>



*)

METHOD lsbIsSet
VAR_INPUT
	(* current value to check *)
	currentValue	:DWORD;
	(* message if the assertion is false *)
	message			:AssertMessage;
END_VAR
IF (NOT TO_BOOL(currentValue AND THIS^.LSB)) THEN
	THIS^.assertionWasWrong(message, THIS^.getDebugInfo('lsbIsSet'));
END_IF
END_METHOD

(*

## Short summary
This assertion method checks if the least significant bit of current value
is unset

.. <legal notes>

legal notes
=================
| SPDX-FileCopyrightText: © 2022 ekvip automation GmbH <info@ekvip.de>
| SPDX-License-Identifier: Apache-2.0
| For details check: Apache-2.0_

.. _Apache-2.0: https://www.apache.org/licenses/LICENSE-2.0

.. </legal notes>



*)

METHOD lsbIsUnset
VAR_INPUT
	(* current value to check *)
	currentValue	:DWORD;
	(* message if the assertion is false *)
	message			:AssertMessage;
END_VAR
IF (TO_BOOL(currentValue AND THIS^.LSB)) THEN
	THIS^.assertionWasWrong(message, THIS^.getDebugInfo('lsbIsUnset'));
END_IF
END_METHOD

(*

## Short summary
This assertion method checks if the most significant bit of current value
is equal to the expected value

.. <legal notes>

legal notes
=================
| SPDX-FileCopyrightText: © 2022 ekvip automation GmbH <info@ekvip.de>
| SPDX-License-Identifier: Apache-2.0
| For details check: Apache-2.0_

.. _Apache-2.0: https://www.apache.org/licenses/LICENSE-2.0

.. </legal notes>



*)

METHOD msbIsEqualTo
VAR_INPUT
	(* current value to check *)
	currentValue	:DWORD;
	(* expected value of msb *)
	expectedValue	:BOOL;
	(* message if the assertion is false *)
	message			:AssertMessage;
END_VAR
IF (TO_BOOL(currentValue AND THIS^.MSB) <> expectedValue) THEN
	THIS^.assertionWasWrong(message, THIS^.getDebugInfo('msbIsEqualTo'));
END_IF
END_METHOD

(*

## Short summary
This assertion method checks if the most significant bit of current value
is not equal to the unexpected value

.. <legal notes>

legal notes
=================
| SPDX-FileCopyrightText: © 2022 ekvip automation GmbH <info@ekvip.de>
| SPDX-License-Identifier: Apache-2.0
| For details check: Apache-2.0_

.. _Apache-2.0: https://www.apache.org/licenses/LICENSE-2.0

.. </legal notes>



*)

METHOD msbIsNotEqualTo
VAR_INPUT
	(* current value to check *)
	currentValue	:DWORD;
	(* unexpected value of msb *)
	unexpectedValue	:BOOL;
	(* message if the assertion is false *)
	message			:AssertMessage;
END_VAR
IF (TO_BOOL(currentValue AND THIS^.MSB) = unexpectedValue) THEN
	THIS^.assertionWasWrong(message, THIS^.getDebugInfo('msbIsNotEqualTo'));
END_IF
END_METHOD

(*

## Short summary
This assertion method checks if the most significant bit of current value
is set

.. <legal notes>

legal notes
=================
| SPDX-FileCopyrightText: © 2022 ekvip automation GmbH <info@ekvip.de>
| SPDX-License-Identifier: Apache-2.0
| For details check: Apache-2.0_

.. _Apache-2.0: https://www.apache.org/licenses/LICENSE-2.0

.. </legal notes>



*)

METHOD msbIsSet
VAR_INPUT
	(* current value to check *)
	currentValue	:DWORD;
	(* message if the assertion is false *)
	message			:AssertMessage;
END_VAR
IF (NOT TO_BOOL(currentValue AND THIS^.MSB)) THEN
	THIS^.assertionWasWrong(message, THIS^.getDebugInfo('msbIsSet'));
END_IF
END_METHOD

(*

## Short summary
This assertion method checks if the most significant bit of current value
is unset

.. <legal notes>

legal notes
=================
| SPDX-FileCopyrightText: © 2022 ekvip automation GmbH <info@ekvip.de>
| SPDX-License-Identifier: Apache-2.0
| For details check: Apache-2.0_

.. _Apache-2.0: https://www.apache.org/licenses/LICENSE-2.0

.. </legal notes>



*)

METHOD msbIsUnset
VAR_INPUT
	(* current value to check *)
	currentValue	:DWORD;
	(* message if the assertion is false *)
	message			:AssertMessage;
END_VAR
IF (TO_BOOL(currentValue AND THIS^.MSB)) THEN
	THIS^.assertionWasWrong(message, THIS^.getDebugInfo('msbIsUnset'));
END_IF
END_METHOD

(*

## Short summary
This assertion method checks if the result current value bitwise ``OR`` mask is equal to the expected value

.. <legal notes>

legal notes
=================
| SPDX-FileCopyrightText: © 2022 ekvip automation GmbH <info@ekvip.de>
| SPDX-License-Identifier: Apache-2.0
| For details check: Apache-2.0_

.. _Apache-2.0: https://www.apache.org/licenses/LICENSE-2.0

.. </legal notes>



*)

METHOD orMaskIsEqualTo
VAR_INPUT
	(* current value to check *)
	currentValue	:DWORD;
	(* 2nd operand for bitwise operation *)
	mask			:DWORD;
	(* expected result after masking *)
	expectedValue	:DWORD;
	(* message if the assertion is false *)
	message			:AssertMessage;
END_VAR
IF ((currentValue OR mask) <> expectedValue) THEN
	THIS^.assertionWasWrong(message, THIS^.getDebugInfo('orMaskIsEqualTo'));
END_IF
END_METHOD

(*

## Short summary
This assertion method checks if the result current value bitwise ``OR`` mask 
is not equal to the unexpected value

.. <legal notes>

legal notes
=================
| SPDX-FileCopyrightText: © 2022 ekvip automation GmbH <info@ekvip.de>
| SPDX-License-Identifier: Apache-2.0
| For details check: Apache-2.0_

.. _Apache-2.0: https://www.apache.org/licenses/LICENSE-2.0

.. </legal notes>



*)

METHOD orMaskIsNotEqualTo
VAR_INPUT
	(* current value to check *)
	currentValue	:DWORD;
	(* 2nd operand for bitwise operation *)
	mask			:DWORD;
	(* unexpected result after masking *)
	unexpectedValue	:DWORD;
	(* message if the assertion is false *)
	message			:AssertMessage;
END_VAR
IF ((currentValue OR mask) = unexpectedValue) THEN
	THIS^.assertionWasWrong(message, THIS^.getDebugInfo('orMaskIsNotEqualTo'));
END_IF
END_METHOD

(*

## Short summary
This assertion method checks if the current value is equal to the expected value

.. <legal notes>

legal notes
=================
| SPDX-FileCopyrightText: © 2022 ekvip automation GmbH <info@ekvip.de>
| SPDX-License-Identifier: Apache-2.0
| For details check: Apache-2.0_

